LIN {X -0.362,Y -583.040,Z 935.630,A 0.000,B 0.000,C 90.000,E1 149.410} C_DIS
LIN {X -0.117,Y -588.452,Z 935.622,A 0.000,B 0.000,C 90.000,E1 148.043} C_DIS
LIN {X 0.030,Y -592.572,Z 935.617,A 0.000,B 0.000,C 90.000,E1 146.962} C_DIS
LIN {X 0.227,Y -596.675,Z 935.611,A 0.000,B 0.000,C 90.000,E1 145.881} C_DIS
LIN {X 0.218,Y -601.491,Z 935.603,A 0.000,B 0.000,C 90.000,E1 144.562} C_DIS
LIN {X -0.105,Y -605.216,Z 935.597,A 0.000,B 0.000,C 90.000,E1 143.543} C_DIS
LIN {X -0.187,Y -610.766,Z 935.589,A 0.000,B 0.000,C 90.000,E1 141.984} C_DIS
LIN {X -0.091,Y -615.489,Z 935.582,A 0.000,B 0.000,C 90.000,E1 140.678} C_DIS
LIN {X 0.004,Y -620.250,Z 935.574,A 0.000,B 0.000,C 90.000,E1 139.380} C_DIS
LIN {X 0.191,Y -624.987,Z 935.567,A 0.000,B 0.000,C 90.000,E1 138.081} C_DIS
LIN {X 0.103,Y -633.010,Z 935.556,A 0.000,B 0.000,C 90.000,E1 136.053} C_DIS
LIN {X -0.067,Y -638.812,Z 935.548,A 0.000,B 0.000,C 90.000,E1 134.555} C_DIS
LIN {X -0.121,Y -644.569,Z 935.539,A 0.000,B 0.000,C 90.000,E1 133.056} C_DIS
LIN {X -0.071,Y -651.286,Z 935.530,A 0.000,B 0.000,C 90.000,E1 131.310} C_DIS
LIN {X -0.269,Y -656.035,Z 935.523,A 0.000,B 0.000,C 90.000,E1 130.092} C_DIS
LIN {X 0.143,Y -662.595,Z 935.513,A 0.000,B 0.000,C 90.000,E1 128.338} C_DIS
LIN {X -0.301,Y -667.183,Z 935.506,A 0.000,B 0.000,C 90.000,E1 127.156} C_DIS
LIN {X -0.153,Y -671.681,Z 935.500,A 0.000,B 0.000,C 90.000,E1 125.931} C_DIS
LIN {X 0.096,Y -674.267,Z 935.496,A 0.000,B 0.000,C 90.000,E1 125.185} C_DIS
LIN {X -0.032,Y -678.225,Z 935.489,A 0.000,B 0.000,C 90.000,E1 123.992} C_DIS
LIN {X -0.273,Y -680.447,Z 935.485,A 0.000,B 0.000,C 90.000,E1 123.293} C_DIS
LIN {X -0.309,Y -683.103,Z 935.480,A 0.000,B 0.000,C 90.000,E1 122.339} C_DIS
LIN {X 0.065,Y -684.898,Z 935.476,A 0.000,B 0.000,C 90.000,E1 121.592} C_DIS
LIN {X -0.272,Y -687.033,Z 935.470,A 0.000,B 0.000,C 90.000,E1 120.669} C_DIS
LIN {X 0.137,Y -688.460,Z 935.466,A 0.000,B 0.000,C 90.000,E1 119.922} C_DIS
LIN {X -0.157,Y -690.099,Z 935.461,A 0.000,B 0.000,C 90.000,E1 118.999} C_DIS
LIN {X 0.309,Y -690.840,Z 935.458,A 0.000,B 0.000,C 90.000,E1 118.487} C_DIS
LIN {X -0.282,Y -691.955,Z 935.453,A 0.000,B 0.000,C 90.000,E1 117.590} C_DIS
LIN {X 0.076,Y -692.662,Z 935.448,A 0.000,B 0.000,C 90.000,E1 116.616} C_DIS
LIN {X 0.133,Y -692.971,Z 935.443,A 0.000,B 0.000,C 90.000,E1 115.668} C_DIS
LIN {X 0.198,Y -693.012,Z 935.437,A 0.000,B 0.000,C 90.000,E1 114.719} C_DIS
LIN {X 0.017,Y -692.878,Z 935.434,A 0.000,B 0.000,C 90.000,E1 114.027} C_DIS
LIN {X 0.261,Y -692.673,Z 935.432,A 0.000,B 0.000,C 90.000,E1 113.770} C_DIS
LIN {X -0.167,Y -691.954,Z 935.430,A 0.000,B 0.000,C 90.000,E1 113.334} C_DIS
LIN {X 0.072,Y -691.188,Z 935.428,A 0.000,B 0.000,C 90.000,E1 113.078} C_DIS
LIN {X 0.307,Y -690.243,Z 935.427,A 0.000,B 0.000,C 90.000,E1 112.823} C_DIS
LIN {X 0.273,Y -689.103,Z 935.426,A 0.000,B 0.000,C 90.000,E1 112.589} C_DIS
LIN {X -0.135,Y -686.943,Z 935.424,A 0.000,B 0.000,C 90.000,E1 112.386} C_DIS
LIN {X -0.277,Y -685.755,Z 935.424,A 0.000,B 0.000,C 90.000,E1 112.280} C_DIS
LIN {X 0.059,Y -682.964,Z 935.422,A 0.000,B 0.000,C 90.000,E1 112.025} C_DIS
LIN {X 0.274,Y -681.246,Z 935.422,A 0.000,B 0.000,C 90.000,E1 111.897} C_DIS
LIN {X -0.208,Y -678.934,Z 935.421,A 0.000,B 0.000,C 90.000,E1 111.844} C_DIS
LIN {X 0.195,Y -676.175,Z 935.421,A 0.000,B 0.000,C 90.000,E1 111.716} C_DIS
LIN {X 0.326,Y -671.403,Z 935.420,A 0.000,B 0.000,C 90.000,E1 111.589} C_DIS
LIN {X 0.190,Y -668.015,Z 935.420,A 0.000,B 0.000,C 90.000,E1 111.535} C_DIS
LIN {X -0.330,Y -660.119,Z 935.420,A 0.000,B 0.000,C 90.000,E1 111.535} C_DIS
LIN {X -0.363,Y -639.191,Z 935.419,A 0.000,B 0.000,C 90.000,E1 111.535} C_DIS
LIN {X 0.038,Y -634.303,Z 935.419,A 0.000,B 0.000,C 90.000,E1 111.461} C_DIS
LIN {X -0.248,Y -628.865,Z 935.419,A 0.000,B 0.000,C 90.000,E1 111.408} C_DIS
LIN {X 0.128,Y -621.355,Z 935.418,A 0.000,B 0.000,C 90.000,E1 111.227} C_DIS
LIN {X 0.020,Y -614.885,Z 935.417,A 0.000,B 0.000,C 90.000,E1 111.046} C_DIS
LIN {X -0.101,Y -607.904,Z 935.416,A 0.000,B 0.000,C 90.000,E1 110.791} C_DIS
LIN {X -0.152,Y -602.249,Z 935.414,A 0.000,B 0.000,C 90.000,E1 110.536} C_DIS
LIN {X 0.285,Y -595.632,Z 935.412,A 0.000,B 0.000,C 90.000,E1 110.120} C_DIS
LIN {X -0.258,Y -586.968,Z 935.409,A 0.000,B 0.000,C 90.000,E1 109.577} C_DIS
LIN {X 0.123,Y -577.996,Z 935.405,A 0.000,B 0.000,C 90.000,E1 108.906} C_DIS
LIN {X -0.168,Y -569.590,Z 935.403,A 0.000,B 0.000,C 90.000,E1 108.471} C_DIS
LIN {X 0.206,Y -564.053,Z 935.401,A 0.000,B 0.000,C 90.000,E1 108.181} C_DIS
LIN {X -0.172,Y -558.813,Z 935.400,A 0.000,B 0.000,C 90.000,E1 108.000} C_DIS
LIN {X 0.052,Y -554.272,Z 935.399,A 0.000,B 0.000,C 90.000,E1 107.764} C_DIS
LIN {X 0.127,Y -552.298,Z 935.398,A 0.000,B 0.000,C 90.000,E1 107.583} C_DIS
LIN {X 0.089,Y -552.284,Z 935.398,A 0.000,B 0.000,C 90.000,E1 107.583} C_DIS
LIN {X -0.183,Y -551.902,Z 935.397,A 0.000,B 0.000,C 90.000,E1 107.402} C_DIS
LIN {X 0.198,Y -552.578,Z 935.387,A 0.000,B 0.000,C 90.000,E1 105.552} C_DIS
LIN {X 0.228,Y -553.493,Z 935.376,A 0.000,B 0.000,C 90.000,E1 103.592} C_DIS
LIN {X 0.150,Y -554.878,Z 935.363,A 0.000,B 0.000,C 90.000,E1 101.366} C_DIS
LIN {X -0.122,Y -556.475,Z 935.352,A 0.000,B 0.000,C 90.000,E1 99.443} C_DIS
LIN {X 0.047,Y -557.835,Z 935.343,A 0.000,B 0.000,C 90.000,E1 97.757} C_DIS
LIN {X 0.020,Y -558.827,Z 935.335,A 0.000,B 0.000,C 90.000,E1 96.372} C_DIS
LIN {X -0.047,Y -559.704,Z 935.328,A 0.000,B 0.000,C 90.000,E1 94.992} C_DIS
LIN {X -0.006,Y -560.667,Z 935.319,A 0.000,B 0.000,C 90.000,E1 93.326} C_DIS
LIN {X -0.166,Y -561.192,Z 935.312,A 0.000,B 0.000,C 90.000,E1 92.236} C_DIS
LIN {X -0.226,Y -561.817,Z 935.305,A 0.000,B 0.000,C 90.000,E1 90.859} C_DIS
LIN {X 0.174,Y -562.176,Z 935.299,A 0.000,B 0.000,C 90.000,E1 89.714} C_DIS
LIN {X 0.114,Y -562.543,Z 935.291,A 0.000,B 0.000,C 90.000,E1 88.339} C_DIS
LIN {X 0.072,Y -562.878,Z 935.283,A 0.000,B 0.000,C 90.000,E1 86.963} C_DIS
LIN {X -0.254,Y -563.186,Z 935.272,A 0.000,B 0.000,C 90.000,E1 85.065} C_DIS
LIN {X -0.244,Y -563.359,Z 935.265,A 0.000,B 0.000,C 90.000,E1 83.685} C_DIS
LIN {X -0.175,Y -563.591,Z 935.257,A 0.000,B 0.000,C 90.000,E1 82.299} C_DIS
LIN {X 0.054,Y -564.071,Z 935.248,A 0.000,B 0.000,C 90.000,E1 80.622} C_DIS
LIN {X 0.152,Y -564.952,Z 935.236,A 0.000,B 0.000,C 90.000,E1 78.409} C_DIS
LIN {X -0.203,Y -566.027,Z 935.225,A 0.000,B 0.000,C 90.000,E1 76.520} C_DIS
LIN {X -0.077,Y -566.750,Z 935.219,A 0.000,B 0.000,C 90.000,E1 75.408} C_DIS
LIN {X 0.137,Y -567.695,Z 935.210,A 0.000,B 0.000,C 90.000,E1 73.740} C_DIS
LIN {X -0.175,Y -568.620,Z 935.201,A 0.000,B 0.000,C 90.000,E1 72.127} C_DIS
LIN {X 0.043,Y -569.522,Z 935.190,A 0.000,B 0.000,C 90.000,E1 70.188} C_DIS
LIN {X 0.125,Y -570.063,Z 935.181,A 0.000,B 0.000,C 90.000,E1 68.539} C_DIS
LIN {X 0.249,Y -570.504,Z 935.170,A 0.000,B 0.000,C 90.000,E1 66.613} C_DIS
LIN {X 0.085,Y -570.711,Z 935.164,A 0.000,B 0.000,C 90.000,E1 65.537} C_DIS
LIN {X -0.070,Y -570.859,Z 935.158,A 0.000,B 0.000,C 90.000,E1 64.460} C_DIS
LIN {X -0.227,Y -571.063,Z 935.152,A 0.000,B 0.000,C 90.000,E1 63.384} C_DIS
LIN {X 0.211,Y -571.167,Z 935.144,A 0.000,B 0.000,C 90.000,E1 61.975} C_DIS
LIN {X 0.247,Y -571.113,Z 935.135,A 0.000,B 0.000,C 90.000,E1 60.333} C_DIS
LIN {X -0.038,Y -571.169,Z 935.128,A 0.000,B 0.000,C 90.000,E1 58.997} C_DIS
LIN {X -0.267,Y -571.086,Z 935.123,A 0.000,B 0.000,C 90.000,E1 58.201} C_DIS
LIN {X -0.310,Y -570.565,Z 935.113,A 0.000,B 0.000,C 90.000,E1 56.294} C_DIS
LIN {X 0.015,Y -569.854,Z 935.105,A 0.000,B 0.000,C 90.000,E1 54.895} C_DIS
LIN {X -0.133,Y -569.057,Z 935.097,A 0.000,B 0.000,C 90.000,E1 53.543} C_DIS
LIN {X -0.094,Y -568.344,Z 935.093,A 0.000,B 0.000,C 90.000,E1 52.718} C_DIS
LIN {X -0.174,Y -567.529,Z 935.088,A 0.000,B 0.000,C 90.000,E1 51.904} C_DIS
LIN {X -0.139,Y -566.224,Z 935.082,A 0.000,B 0.000,C 90.000,E1 50.803} C_DIS
LIN {X -0.237,Y -565.126,Z 935.078,A 0.000,B 0.000,C 90.000,E1 49.989} C_DIS
LIN {X 0.344,Y -564.350,Z 935.075,A 0.000,B 0.000,C 90.000,E1 49.380} C_DIS
LIN {X -0.201,Y -562.938,Z 935.070,A 0.000,B 0.000,C 90.000,E1 48.609} C_DIS
LIN {X 0.125,Y -560.668,Z 935.064,A 0.000,B 0.000,C 90.000,E1 47.472} C_DIS
LIN {X -0.124,Y -559.464,Z 935.061,A 0.000,B 0.000,C 90.000,E1 46.944} C_DIS
LIN {X 0.117,Y -556.574,Z 935.055,A 0.000,B 0.000,C 90.000,E1 45.810} C_DIS
LIN {X -0.221,Y -555.832,Z 935.053,A 0.000,B 0.000,C 90.000,E1 45.567} C_DIS
LIN {X -0.027,Y -552.309,Z 935.047,A 0.000,B 0.000,C 90.000,E1 44.433} C_DIS
LIN {X 0.007,Y -551.392,Z 935.045,A 0.000,B 0.000,C 90.000,E1 44.150} C_DIS
LIN {X 0.109,Y -548.247,Z 935.041,A 0.000,B 0.000,C 90.000,E1 43.299} C_DIS
LIN {X -0.220,Y -546.013,Z 935.038,A 0.000,B 0.000,C 90.000,E1 42.771} C_DIS
LIN {X 0.002,Y -542.942,Z 935.034,A 0.000,B 0.000,C 90.000,E1 42.043} C_DIS
LIN {X 0.230,Y -539.518,Z 935.030,A 0.000,B 0.000,C 90.000,E1 41.310} C_DIS
LIN {X -0.153,Y -536.559,Z 935.027,A 0.000,B 0.000,C 90.000,E1 40.782} C_DIS
LIN {X 0.198,Y -533.440,Z 935.023,A 0.000,B 0.000,C 90.000,E1 40.172} C_DIS
LIN {X -0.225,Y -530.096,Z 935.020,A 0.000,B 0.000,C 90.000,E1 39.644} C_DIS
LIN {X 0.010,Y -523.010,Z 935.014,A 0.000,B 0.000,C 90.000,E1 38.463} C_DIS
LIN {X 0.059,Y -518.243,Z 935.010,A 0.000,B 0.000,C 90.000,E1 37.729} C_DIS
LIN {X -0.127,Y -512.183,Z 935.005,A 0.000,B 0.000,C 90.000,E1 36.870} C_DIS
LIN {X 0.229,Y -506.756,Z 935.001,A 0.000,B 0.000,C 90.000,E1 36.091} C_DIS
LIN {X -0.065,Y -503.303,Z 934.998,A 0.000,B 0.000,C 90.000,E1 35.678} C_DIS
LIN {X 0.155,Y -500.020,Z 934.996,A 0.000,B 0.000,C 90.000,E1 35.231} C_DIS
LIN {X 0.123,Y -493.520,Z 934.992,A 0.000,B 0.000,C 90.000,E1 34.485} C_DIS
LIN {X 0.010,Y -490.928,Z 934.990,A 0.000,B 0.000,C 90.000,E1 34.199} C_DIS
LIN {X -0.230,Y -483.914,Z 934.986,A 0.000,B 0.000,C 90.000,E1 33.499} C_DIS
LIN {X 0.225,Y -478.200,Z 934.983,A 0.000,B 0.000,C 90.000,E1 32.880} C_DIS
LIN {X 0.050,Y -470.972,Z 934.979,A 0.000,B 0.000,C 90.000,E1 32.212} C_DIS
LIN {X 0.072,Y -460.714,Z 934.974,A 0.000,B 0.000,C 90.000,E1 31.288} C_DIS
LIN {X -0.009,Y -450.031,Z 934.969,A 0.000,B 0.000,C 90.000,E1 30.384} C_DIS
LIN {X 0.134,Y -437.697,Z 934.963,A 0.000,B 0.000,C 90.000,E1 29.333} C_DIS
LIN {X 0.113,Y -416.401,Z 934.953,A 0.000,B 0.000,C 90.000,E1 27.462} C_DIS
LIN {X -0.085,Y -400.384,Z 934.944,A 0.000,B 0.000,C 90.000,E1 25.924} C_DIS
LIN {X 0.089,Y -397.514,Z 934.942,A 0.000,B 0.000,C 90.000,E1 25.591} C_DIS
LIN {X -0.048,Y -393.296,Z 934.939,A 0.000,B 0.000,C 90.000,E1 25.027} C_DIS
LIN {X -0.019,Y -390.739,Z 934.936,A 0.000,B 0.000,C 90.000,E1 24.515} C_DIS
LIN {X -0.019,Y -389.495,Z 934.934,A 0.000,B 0.000,C 90.000,E1 24.027} C_DIS
LIN {X 0.106,Y -388.958,Z 934.929,A 0.000,B 0.000,C 90.000,E1 23.206} C_DIS
LIN {X -0.027,Y -389.146,Z 934.924,A 0.000,B 0.000,C 90.000,E1 22.333} C_DIS
LIN {X -0.081,Y -392.397,Z 934.904,A 0.000,B 0.000,C 90.000,E1 18.779} C_DIS
LIN {X 0.180,Y -395.235,Z 934.891,A 0.000,B 0.000,C 90.000,E1 16.260} C_DIS
LIN {X -0.033,Y -399.362,Z 934.873,A 0.000,B 0.000,C 90.000,E1 13.119} C_DIS
LIN {X 0.028,Y -403.553,Z 934.857,A 0.000,B 0.000,C 90.000,E1 10.310} C_DIS
LIN {X 0.037,Y -405.864,Z 934.850,A 0.000,B 0.000,C 90.000,E1 8.916} C_DIS
LIN {X 0.060,Y -409.516,Z 934.838,A 0.000,B 0.000,C 90.000,E1 6.834} C_DIS
LIN {X 0.117,Y -414.812,Z 934.823,A 0.000,B 0.000,C 90.000,E1 4.073} C_DIS
LIN {X -0.069,Y -421.450,Z 934.806,A 0.000,B 0.000,C 90.000,E1 1.031} C_DIS
LIN {X -0.163,Y -426.045,Z 934.795,A 0.000,B 0.000,C 90.000,E1 359.141} C_DIS
LIN {X -0.053,Y -427.988,Z 934.791,A 0.000,B 0.000,C 90.000,E1 358.453} C_DIS
LIN {X 0.173,Y -430.450,Z 934.788,A 0.000,B 0.000,C 90.000,E1 357.764} C_DIS
LIN {X 0.208,Y -431.327,Z 934.787,A 0.000,B 0.000,C 90.000,E1 357.593} C_DIS
LIN {X -0.150,Y -433.776,Z 934.785,A 0.000,B 0.000,C 90.000,E1 357.306} C_DIS
LIN {X 0.127,Y -435.457,Z 934.784,A 0.000,B 0.000,C 90.000,E1 357.020} C_DIS
LIN {X -0.069,Y -436.183,Z 934.783,A 0.000,B 0.000,C 90.000,E1 356.963} C_DIS
LIN {X -0.052,Y -441.451,Z 934.781,A 0.000,B 0.000,C 90.000,E1 356.560} C_DIS
LIN {X 0.217,Y -447.579,Z 934.779,A 0.000,B 0.000,C 90.000,E1 356.216} C_DIS
LIN {X 0.059,Y -454.281,Z 934.777,A 0.000,B 0.000,C 90.000,E1 355.927} C_DIS
LIN {X 0.204,Y -467.603,Z 934.774,A 0.000,B 0.000,C 90.000,E1 355.241} C_DIS
LIN {X 0.040,Y -482.471,Z 934.769,A 0.000,B 0.000,C 90.000,E1 354.489} C_DIS
LIN {X -0.188,Y -490.646,Z 934.767,A 0.000,B 0.000,C 90.000,E1 354.090} C_DIS
LIN {X 0.143,Y -503.360,Z 934.763,A 0.000,B 0.000,C 90.000,E1 353.337} C_DIS
LIN {X 0.162,Y -512.995,Z 934.760,A 0.000,B 0.000,C 90.000,E1 352.761} C_DIS
LIN {X -0.105,Y -522.411,Z 934.757,A 0.000,B 0.000,C 90.000,E1 352.186} C_DIS
LIN {X 0.229,Y -528.534,Z 934.754,A 0.000,B 0.000,C 90.000,E1 351.724} C_DIS
LIN {X -0.112,Y -535.939,Z 934.751,A 0.000,B 0.000,C 90.000,E1 351.197} C_DIS
LIN {X -0.284,Y -543.099,Z 934.748,A 0.000,B 0.000,C 90.000,E1 350.622} C_DIS
LIN {X -0.120,Y -549.902,Z 934.744,A 0.000,B 0.000,C 90.000,E1 349.982} C_DIS
LIN {X -0.031,Y -555.068,Z 934.741,A 0.000,B 0.000,C 90.000,E1 349.454} C_DIS
LIN {X 0.254,Y -561.010,Z 934.738,A 0.000,B 0.000,C 90.000,E1 348.757} C_DIS
LIN {X 0.045,Y -568.927,Z 934.732,A 0.000,B 0.000,C 90.000,E1 347.813} C_DIS
LIN {X 0.167,Y -573.969,Z 934.729,A 0.000,B 0.000,C 90.000,E1 347.117} C_DIS
LIN {X 0.219,Y -579.696,Z 934.724,A 0.000,B 0.000,C 90.000,E1 346.297} C_DIS
LIN {X -0.001,Y -583.991,Z 934.720,A 0.000,B 0.000,C 90.000,E1 345.644} C_DIS
LIN {X 0.301,Y -588.909,Z 934.716,A 0.000,B 0.000,C 90.000,E1 344.810} C_DIS
LIN {X -0.146,Y -594.211,Z 934.711,A 0.000,B 0.000,C 90.000,E1 343.921} C_DIS
LIN {X -0.028,Y -599.726,Z 934.705,A 0.000,B 0.000,C 90.000,E1 342.851} C_DIS
LIN {X -0.052,Y -608.018,Z 934.695,A 0.000,B 0.000,C 90.000,E1 341.148} C_DIS
LIN {X -0.108,Y -612.243,Z 934.690,A 0.000,B 0.000,C 90.000,E1 340.242} C_DIS
LIN {X -0.176,Y -617.810,Z 934.683,A 0.000,B 0.000,C 90.000,E1 338.954} C_DIS
LIN {X -0.155,Y -622.956,Z 934.676,A 0.000,B 0.000,C 90.000,E1 337.667} C_DIS
LIN {X 0.171,Y -625.871,Z 934.672,A 0.000,B 0.000,C 90.000,E1 336.869} C_DIS
LIN {X -0.037,Y -629.434,Z 934.666,A 0.000,B 0.000,C 90.000,E1 335.869} C_DIS
LIN {X 0.034,Y -632.073,Z 934.662,A 0.000,B 0.000,C 90.000,E1 335.101} C_DIS
LIN {X 0.181,Y -635.351,Z 934.656,A 0.000,B 0.000,C 90.000,E1 334.076} C_DIS
LIN {X 0.141,Y -639.086,Z 934.649,A 0.000,B 0.000,C 90.000,E1 332.820} C_DIS
LIN {X -0.192,Y -641.900,Z 934.644,A 0.000,B 0.000,C 90.000,E1 331.847} C_DIS
LIN {X -0.177,Y -644.440,Z 934.638,A 0.000,B 0.000,C 90.000,E1 330.845} C_DIS
LIN {X 0.042,Y -647.954,Z 934.630,A 0.000,B 0.000,C 90.000,E1 329.331} C_DIS
LIN {X 0.148,Y -650.027,Z 934.624,A 0.000,B 0.000,C 90.000,E1 328.329} C_DIS
LIN {X -0.271,Y -651.825,Z 934.619,A 0.000,B 0.000,C 90.000,E1 327.375} C_DIS
LIN {X -0.209,Y -653.092,Z 934.615,A 0.000,B 0.000,C 90.000,E1 326.628} C_DIS
LIN {X 0.314,Y -654.556,Z 934.609,A 0.000,B 0.000,C 90.000,E1 325.595} C_DIS
LIN {X 0.327,Y -656.333,Z 934.601,A 0.000,B 0.000,C 90.000,E1 324.116} C_DIS
LIN {X 0.354,Y -657.418,Z 934.595,A 0.000,B 0.000,C 90.000,E1 323.130} C_DIS
LIN {X -0.117,Y -658.660,Z 934.587,A 0.000,B 0.000,C 90.000,E1 321.698} C_DIS
LIN {X -0.230,Y -660.230,Z 934.576,A 0.000,B 0.000,C 90.000,E1 319.747} C_DIS
LIN {X 0.161,Y -661.603,Z 934.567,A 0.000,B 0.000,C 90.000,E1 318.000} C_DIS
LIN {X 0.130,Y -662.427,Z 934.561,A 0.000,B 0.000,C 90.000,E1 317.025} C_DIS
LIN {X 0.063,Y -663.474,Z 934.555,A 0.000,B 0.000,C 90.000,E1 315.810} C_DIS
LIN {X -0.018,Y -665.725,Z 934.540,A 0.000,B 0.000,C 90.000,E1 313.137} C_DIS
LIN {X -0.002,Y -667.109,Z 934.532,A 0.000,B 0.000,C 90.000,E1 311.676} C_DIS
LIN {X 0.115,Y -668.674,Z 934.522,A 0.000,B 0.000,C 90.000,E1 309.967} C_DIS
LIN {X 0.185,Y -669.760,Z 934.515,A 0.000,B 0.000,C 90.000,E1 308.749} C_DIS
LIN {X -0.163,Y -670.700,Z 934.509,A 0.000,B 0.000,C 90.000,E1 307.569} C_DIS
LIN {X 0.044,Y -671.266,Z 934.503,A 0.000,B 0.000,C 90.000,E1 306.583} C_DIS
LIN {X -0.258,Y -671.525,Z 934.499,A 0.000,B 0.000,C 90.000,E1 305.884} C_DIS
LIN {X -0.326,Y -672.092,Z 934.490,A 0.000,B 0.000,C 90.000,E1 304.199} C_DIS
LIN {X -0.084,Y -673.147,Z 934.478,A 0.000,B 0.000,C 90.000,E1 302.005} C_DIS
LIN {X -0.300,Y -678.749,Z 934.447,A 0.000,B 0.000,C 90.000,E1 296.488} C_DIS
LIN {X -0.219,Y -680.724,Z 934.440,A 0.000,B 0.000,C 90.000,E1 295.283} C_DIS
LIN {X -0.106,Y -682.529,Z 934.434,A 0.000,B 0.000,C 90.000,E1 294.079} C_DIS
LIN {X 0.238,Y -683.405,Z 934.430,A 0.000,B 0.000,C 90.000,E1 293.334} C_DIS
LIN {X -0.184,Y -683.659,Z 934.428,A 0.000,B 0.000,C 90.000,E1 293.131} C_DIS
LIN {X -0.037,Y -683.885,Z 934.426,A 0.000,B 0.000,C 90.000,E1 292.642} C_DIS
LIN {X 0.168,Y -683.807,Z 934.424,A 0.000,B 0.000,C 90.000,E1 292.386} C_DIS
LIN {X 0.318,Y -683.227,Z 934.422,A 0.000,B 0.000,C 90.000,E1 291.897} C_DIS
LIN {X -0.367,Y -682.487,Z 934.421,A 0.000,B 0.000,C 90.000,E1 291.716} C_DIS
LIN {X -0.266,Y -681.729,Z 934.420,A 0.000,B 0.000,C 90.000,E1 291.589} C_DIS
LIN {X -0.127,Y -677.804,Z 934.417,A 0.000,B 0.000,C 90.000,E1 291.099} C_DIS
LIN {X -0.035,Y -676.505,Z 934.417,A 0.000,B 0.000,C 90.000,E1 290.972} C_DIS
LIN {X 0.005,Y -669.890,Z 934.414,A 0.000,B 0.000,C 90.000,E1 290.556} C_DIS
LIN {X 0.263,Y -663.844,Z 934.412,A 0.000,B 0.000,C 90.000,E1 290.174} C_DIS
LIN {X -0.173,Y -662.168,Z 934.411,A 0.000,B 0.000,C 90.000,E1 290.066} C_DIS
LIN {X -0.213,Y -662.151,Z 934.411,A 0.000,B 0.000,C 90.000,E1 290.066} C_DIS
LIN {X -0.036,Y -661.882,Z 934.411,A 0.000,B 0.000,C 90.000,E1 289.939} C_DIS
LIN {X 0.111,Y -661.958,Z 934.410,A 0.000,B 0.000,C 90.000,E1 289.812} C_DIS
LIN {X 0.003,Y -662.374,Z 934.409,A 0.000,B 0.000,C 90.000,E1 289.577} C_DIS
LIN {X 0.118,Y -663.165,Z 934.407,A 0.000,B 0.000,C 90.000,E1 289.322} C_DIS
LIN {X 0.016,Y -664.110,Z 934.406,A 0.000,B 0.000,C 90.000,E1 289.087} C_DIS
LIN {X 0.010,Y -667.041,Z 934.403,A 0.000,B 0.000,C 90.000,E1 288.489} C_DIS
LIN {X 0.037,Y -671.497,Z 934.398,A 0.000,B 0.000,C 90.000,E1 287.638} C_DIS
LIN {X -0.101,Y -673.850,Z 934.395,A 0.000,B 0.000,C 90.000,E1 287.166} C_DIS
LIN {X -0.081,Y -676.901,Z 934.391,A 0.000,B 0.000,C 90.000,E1 286.441} C_DIS
LIN {X -0.041,Y -679.329,Z 934.387,A 0.000,B 0.000,C 90.000,E1 285.717} C_DIS
LIN {X -0.125,Y -680.682,Z 934.385,A 0.000,B 0.000,C 90.000,E1 285.245} C_DIS
LIN {X -0.262,Y -682.869,Z 934.379,A 0.000,B 0.000,C 90.000,E1 284.300} C_DIS
LIN {X -0.320,Y -683.809,Z 934.377,A 0.000,B 0.000,C 90.000,E1 283.828} C_DIS
LIN {X 0.250,Y -685.364,Z 934.371,A 0.000,B 0.000,C 90.000,E1 282.827} C_DIS
LIN {X 0.187,Y -686.270,Z 934.367,A 0.000,B 0.000,C 90.000,E1 282.119} C_DIS
LIN {X 0.008,Y -686.722,Z 934.365,A 0.000,B 0.000,C 90.000,E1 281.658} C_DIS
LIN {X -0.029,Y -686.947,Z 934.362,A 0.000,B 0.000,C 90.000,E1 281.186} C_DIS
LIN {X -0.067,Y -686.915,Z 934.360,A 0.000,B 0.000,C 90.000,E1 280.715} C_DIS
LIN {X -0.233,Y -686.522,Z 934.357,A 0.000,B 0.000,C 90.000,E1 280.254} C_DIS
LIN {X -0.255,Y -686.208,Z 934.356,A 0.000,B 0.000,C 90.000,E1 280.018} C_DIS
LIN {X 0.256,Y -685.292,Z 934.353,A 0.000,B 0.000,C 90.000,E1 279.500} C_DIS
LIN {X 0.197,Y -683.887,Z 934.350,A 0.000,B 0.000,C 90.000,E1 279.029} C_DIS
LIN {X 0.020,Y -682.123,Z 934.348,A 0.000,B 0.000,C 90.000,E1 278.568} C_DIS
LIN {X -0.163,Y -679.996,Z 934.345,A 0.000,B 0.000,C 90.000,E1 278.106} C_DIS
LIN {X 0.181,Y -675.839,Z 934.340,A 0.000,B 0.000,C 90.000,E1 277.239} C_DIS
LIN {X -0.280,Y -670.704,Z 934.335,A 0.000,B 0.000,C 90.000,E1 276.315} C_DIS
LIN {X 0.129,Y -667.800,Z 934.332,A 0.000,B 0.000,C 90.000,E1 275.796} C_DIS
LIN {X -0.146,Y -664.503,Z 934.330,A 0.000,B 0.000,C 90.000,E1 275.334} C_DIS
LIN {X 0.123,Y -659.733,Z 934.326,A 0.000,B 0.000,C 90.000,E1 274.702} C_DIS
LIN {X -0.254,Y -655.607,Z 934.323,A 0.000,B 0.000,C 90.000,E1 274.245} C_DIS
LIN {X -0.060,Y -649.876,Z 934.320,A 0.000,B 0.000,C 90.000,E1 273.612} C_DIS
LIN {X 0.281,Y -645.013,Z 934.317,A 0.000,B 0.000,C 90.000,E1 273.094} C_DIS
LIN {X 0.109,Y -638.445,Z 934.314,A 0.000,B 0.000,C 90.000,E1 272.522} C_DIS
LIN {X 0.273,Y -631.457,Z 934.311,A 0.000,B 0.000,C 90.000,E1 271.949} C_DIS
LIN {X 0.211,Y -624.054,Z 934.308,A 0.000,B 0.000,C 90.000,E1 271.432} C_DIS
LIN {X 0.212,Y -617.936,Z 934.306,A 0.000,B 0.000,C 90.000,E1 271.031} C_DIS
LIN {X -0.205,Y -611.553,Z 934.304,A 0.000,B 0.000,C 90.000,E1 270.688} C_DIS
LIN {X 0.261,Y -604.962,Z 934.302,A 0.000,B 0.000,C 90.000,E1 270.286} C_DIS
LIN {X -0.198,Y -598.161,Z 934.300,A 0.000,B 0.000,C 90.000,E1 270.000} C_DIS
LIN {X 0.219,Y -591.125,Z 934.298,A 0.000,B 0.000,C 90.000,E1 269.656} C_DIS
LIN {X -0.142,Y -585.444,Z 934.297,A 0.000,B 0.000,C 90.000,E1 269.484} C_DIS
LIN {X -0.137,Y -577.860,Z 934.296,A 0.000,B 0.000,C 90.000,E1 269.255} C_DIS
LIN {X -0.221,Y -570.064,Z 934.295,A 0.000,B 0.000,C 90.000,E1 269.083} C_DIS
LIN {X -0.193,Y -563.989,Z 934.294,A 0.000,B 0.000,C 90.000,E1 268.969} C_DIS
LIN {X -0.243,Y -557.682,Z 934.294,A 0.000,B 0.000,C 90.000,E1 268.912} C_DIS
LIN {X -0.093,Y -552.004,Z 934.294,A 0.000,B 0.000,C 90.000,E1 268.854} C_DIS
LIN {X 0.239,Y -550.919,Z 934.294,A 0.000,B 0.000,C 90.000,E1 268.797} C_DIS
LIN {X 0.193,Y -550.707,Z 934.293,A 0.000,B 0.000,C 90.000,E1 268.797} C_DIS
LIN {X -0.185,Y -549.196,Z 934.292,A 0.000,B 0.000,C 90.000,E1 268.625} C_DIS
LIN {X 0.184,Y -545.518,Z 934.290,A 0.000,B 0.000,C 90.000,E1 268.165} C_DIS
LIN {X 0.060,Y -544.029,Z 934.289,A 0.000,B 0.000,C 90.000,E1 268.051} C_DIS
LIN {X 0.017,Y -543.977,Z 934.289,A 0.000,B 0.000,C 90.000,E1 268.051} C_DIS
LIN {X 0.228,Y -543.627,Z 934.288,A 0.000,B 0.000,C 90.000,E1 267.879} C_DIS
LIN {X -0.146,Y -542.881,Z 934.285,A 0.000,B 0.000,C 90.000,E1 267.364} C_DIS
LIN {X 0.213,Y -540.432,Z 934.270,A 0.000,B 0.000,C 90.000,E1 264.489} C_DIS
LIN {X -0.119,Y -539.299,Z 934.260,A 0.000,B 0.000,C 90.000,E1 262.818} C_DIS
LIN {X 0.055,Y -538.331,Z 934.252,A 0.000,B 0.000,C 90.000,E1 261.376} C_DIS
LIN {X 0.249,Y -537.661,Z 934.247,A 0.000,B 0.000,C 90.000,E1 260.500} C_DIS
LIN {X -0.182,Y -536.656,Z 934.243,A 0.000,B 0.000,C 90.000,E1 259.690} C_DIS
LIN {X 0.056,Y -535.034,Z 934.236,A 0.000,B 0.000,C 90.000,E1 258.522} C_DIS
LIN {X 0.172,Y -530.972,Z 934.219,A 0.000,B 0.000,C 90.000,E1 255.353} C_DIS
LIN {X 0.117,Y -528.945,Z 934.209,A 0.000,B 0.000,C 90.000,E1 253.630} C_DIS
LIN {X 0.166,Y -526.789,Z 934.200,A 0.000,B 0.000,C 90.000,E1 251.891} C_DIS
LIN {X -0.163,Y -524.571,Z 934.190,A 0.000,B 0.000,C 90.000,E1 250.188} C_DIS
LIN {X -0.022,Y -522.711,Z 934.182,A 0.000,B 0.000,C 90.000,E1 248.720} C_DIS
LIN {X 0.277,Y -520.814,Z 934.174,A 0.000,B 0.000,C 90.000,E1 247.230} C_DIS
LIN {X 0.204,Y -518.179,Z 934.164,A 0.000,B 0.000,C 90.000,E1 245.485} C_DIS
LIN {X -0.183,Y -515.465,Z 934.154,A 0.000,B 0.000,C 90.000,E1 243.768} C_DIS
LIN {X -0.049,Y -513.030,Z 934.146,A 0.000,B 0.000,C 90.000,E1 242.281} C_DIS
LIN {X 0.038,Y -510.576,Z 934.138,A 0.000,B 0.000,C 90.000,E1 240.795} C_DIS
LIN {X -0.011,Y -508.509,Z 934.131,A 0.000,B 0.000,C 90.000,E1 239.616} C_DIS
LIN {X 0.164,Y -506.356,Z 934.125,A 0.000,B 0.000,C 90.000,E1 238.408} C_DIS
LIN {X -0.120,Y -503.875,Z 934.118,A 0.000,B 0.000,C 90.000,E1 237.248} C_DIS
LIN {X -0.264,Y -499.775,Z 934.108,A 0.000,B 0.000,C 90.000,E1 235.468} C_DIS
LIN {X -0.204,Y -494.327,Z 934.095,A 0.000,B 0.000,C 90.000,E1 233.050} C_DIS
LIN {X -0.235,Y -491.067,Z 934.086,A 0.000,B 0.000,C 90.000,E1 231.537} C_DIS
LIN {X -0.027,Y -487.673,Z 934.078,A 0.000,B 0.000,C 90.000,E1 229.989} C_DIS
LIN {X -0.123,Y -483.469,Z 934.068,A 0.000,B 0.000,C 90.000,E1 228.162} C_DIS
LIN {X 0.131,Y -478.613,Z 934.056,A 0.000,B 0.000,C 90.000,E1 225.972} C_DIS
LIN {X 0.030,Y -475.242,Z 934.047,A 0.000,B 0.000,C 90.000,E1 224.433} C_DIS
LIN {X 0.297,Y -471.084,Z 934.036,A 0.000,B 0.000,C 90.000,E1 222.528} C_DIS
LIN {X 0.070,Y -467.583,Z 934.028,A 0.000,B 0.000,C 90.000,E1 220.987} C_DIS
LIN {X 0.038,Y -462.161,Z 934.014,A 0.000,B 0.000,C 90.000,E1 218.463} C_DIS
LIN {X -0.046,Y -459.386,Z 934.007,A 0.000,B 0.000,C 90.000,E1 217.202} C_DIS
LIN {X 0.015,Y -455.975,Z 933.998,A 0.000,B 0.000,C 90.000,E1 215.598} C_DIS
LIN {X 0.020,Y -452.484,Z 933.989,A 0.000,B 0.000,C 90.000,E1 213.992} C_DIS
LIN {X -0.061,Y -446.698,Z 933.975,A 0.000,B 0.000,C 90.000,E1 211.416} C_DIS
LIN {X -0.171,Y -443.828,Z 933.967,A 0.000,B 0.000,C 90.000,E1 210.129} C_DIS
LIN {X -0.078,Y -439.583,Z 933.956,A 0.000,B 0.000,C 90.000,E1 208.153} C_DIS
LIN {X 0.044,Y -436.809,Z 933.949,A 0.000,B 0.000,C 90.000,E1 206.821} C_DIS
LIN {X -0.039,Y -432.386,Z 933.938,A 0.000,B 0.000,C 90.000,E1 204.847} C_DIS
LIN {X 0.154,Y -428.022,Z 933.927,A 0.000,B 0.000,C 90.000,E1 202.823} C_DIS
LIN {X -0.103,Y -423.545,Z 933.916,A 0.000,B 0.000,C 90.000,E1 200.844} C_DIS
LIN {X 0.146,Y -417.186,Z 933.899,A 0.000,B 0.000,C 90.000,E1 197.764} C_DIS
LIN {X -0.002,Y -413.844,Z 933.889,A 0.000,B 0.000,C 90.000,E1 196.079} C_DIS
LIN {X -0.067,Y -411.056,Z 933.882,A 0.000,B 0.000,C 90.000,E1 194.717} C_DIS
LIN {X 0.066,Y -404.789,Z 933.865,A 0.000,B 0.000,C 90.000,E1 191.591} C_DIS
LIN {X 0.079,Y -401.420,Z 933.855,A 0.000,B 0.000,C 90.000,E1 189.849} C_DIS
LIN {X 0.009,Y -397.329,Z 933.843,A 0.000,B 0.000,C 90.000,E1 187.757} C_DIS
LIN {X -0.150,Y -394.647,Z 933.835,A 0.000,B 0.000,C 90.000,E1 186.372} C_DIS
LIN {X 0.017,Y -388.684,Z 933.818,A 0.000,B 0.000,C 90.000,E1 183.154} C_DIS
LIN {X -0.067,Y -383.430,Z 933.800,A 0.000,B 0.000,C 90.000,E1 179.943} C_DIS
LIN {X -0.016,Y -382.158,Z 933.794,A 0.000,B 0.000,C 90.000,E1 178.854} C_DIS
LIN {X 0.087,Y -381.481,Z 933.789,A 0.000,B 0.000,C 90.000,E1 177.936} C_DIS
LIN {X 0.132,Y -381.508,Z 933.783,A 0.000,B 0.000,C 90.000,E1 176.963} C_DIS
LIN {X -0.090,Y -382.040,Z 933.779,A 0.000,B 0.000,C 90.000,E1 176.274} C_DIS
LIN {X 0.134,Y -383.143,Z 933.776,A 0.000,B 0.000,C 90.000,E1 175.698} C_DIS
LIN {X -0.148,Y -383.539,Z 933.775,A 0.000,B 0.000,C 90.000,E1 175.469} C_DIS
LIN {X -0.074,Y -385.292,Z 933.772,A 0.000,B 0.000,C 90.000,E1 175.008} C_DIS
LIN {X 0.159,Y -388.872,Z 933.769,A 0.000,B 0.000,C 90.000,E1 174.375} C_DIS
LIN {X 0.105,Y -390.089,Z 933.768,A 0.000,B 0.000,C 90.000,E1 174.204} C_DIS
LIN {X -0.173,Y -394.665,Z 933.765,A 0.000,B 0.000,C 90.000,E1 173.742} C_DIS
LIN {X 0.042,Y -401.204,Z 933.762,A 0.000,B 0.000,C 90.000,E1 173.109} C_DIS
LIN {X -0.112,Y -414.286,Z 933.756,A 0.000,B 0.000,C 90.000,E1 172.129} C_DIS
LIN {X -0.098,Y -429.985,Z 933.749,A 0.000,B 0.000,C 90.000,E1 170.905} C_DIS
LIN {X -0.152,Y -439.190,Z 933.745,A 0.000,B 0.000,C 90.000,E1 170.151} C_DIS
LIN {X -0.068,Y -448.118,Z 933.741,A 0.000,B 0.000,C 90.000,E1 169.342} C_DIS
LIN {X 0.255,Y -458.464,Z 933.735,A 0.000,B 0.000,C 90.000,E1 168.342} C_DIS
LIN {X 0.022,Y -466.782,Z 933.731,A 0.000,B 0.000,C 90.000,E1 167.521} C_DIS
LIN {X -0.139,Y -477.531,Z 933.724,A 0.000,B 0.000,C 90.000,E1 166.353} C_DIS
LIN {X 0.080,Y -485.098,Z 933.719,A 0.000,B 0.000,C 90.000,E1 165.408} C_DIS
LIN {X -0.174,Y -492.693,Z 933.714,A 0.000,B 0.000,C 90.000,E1 164.519} C_DIS
LIN {X 0.004,Y -498.226,Z 933.710,A 0.000,B 0.000,C 90.000,E1 163.740} C_DIS
LIN {X 0.031,Y -504.749,Z 933.705,A 0.000,B 0.000,C 90.000,E1 162.834} C_DIS
LIN {X 0.149,Y -516.914,Z 933.695,A 0.000,B 0.000,C 90.000,E1 161.040} C_DIS
LIN {X 0.069,Y -521.689,Z 933.691,A 0.000,B 0.000,C 90.000,E1 160.315} C_DIS
LIN {X 0.059,Y -531.922,Z 933.682,A 0.000,B 0.000,C 90.000,E1 158.720} C_DIS
LIN {X 0.161,Y -537.223,Z 933.677,A 0.000,B 0.000,C 90.000,E1 157.847} C_DIS
LIN {X 0.084,Y -549.262,Z 933.666,A 0.000,B 0.000,C 90.000,E1 155.869} C_DIS
LIN {X 0.106,Y -552.497,Z 933.663,A 0.000,B 0.000,C 90.000,E1 155.305} C_DIS
LIN {X -0.149,Y -559.468,Z 933.656,A 0.000,B 0.000,C 90.000,E1 154.076} C_DIS
LIN {X 0.152,Y -564.538,Z 933.651,A 0.000,B 0.000,C 90.000,E1 153.076} C_DIS
LIN {X 0.176,Y -569.929,Z 933.644,A 0.000,B 0.000,C 90.000,E1 151.975} C_DIS
LIN {X -0.225,Y -575.091,Z 933.638,A 0.000,B 0.000,C 90.000,E1 150.923} C_DIS
LIN {X 0.245,Y -577.525,Z 933.635,A 0.000,B 0.000,C 90.000,E1 150.333} C_DIS
LIN {X -0.063,Y -582.178,Z 933.629,A 0.000,B 0.000,C 90.000,E1 149.282} C_DIS
LIN {X 0.167,Y -587.646,Z 933.622,A 0.000,B 0.000,C 90.000,E1 147.916} C_DIS
LIN {X 0.300,Y -591.804,Z 933.616,A 0.000,B 0.000,C 90.000,E1 146.834} C_DIS
LIN {X -0.008,Y -595.935,Z 933.610,A 0.000,B 0.000,C 90.000,E1 145.801} C_DIS
LIN {X -0.265,Y -599.898,Z 933.604,A 0.000,B 0.000,C 90.000,E1 144.769} C_DIS
LIN {X -0.126,Y -603.663,Z 933.598,A 0.000,B 0.000,C 90.000,E1 143.703} C_DIS
LIN {X -0.145,Y -608.333,Z 933.591,A 0.000,B 0.000,C 90.000,E1 142.396} C_DIS
LIN {X 0.025,Y -614.999,Z 933.581,A 0.000,B 0.000,C 90.000,E1 140.561} C_DIS
LIN {X -0.278,Y -619.806,Z 933.574,A 0.000,B 0.000,C 90.000,E1 139.299} C_DIS
LIN {X 0.045,Y -623.639,Z 933.568,A 0.000,B 0.000,C 90.000,E1 138.243} C_DIS
LIN {X 0.036,Y -630.642,Z 933.558,A 0.000,B 0.000,C 90.000,E1 136.458} C_DIS
LIN {X 0.032,Y -634.670,Z 933.553,A 0.000,B 0.000,C 90.000,E1 135.445} C_DIS
LIN {X -0.104,Y -640.465,Z 933.544,A 0.000,B 0.000,C 90.000,E1 133.947} C_DIS
LIN {X -0.045,Y -645.294,Z 933.537,A 0.000,B 0.000,C 90.000,E1 132.690} C_DIS
LIN {X 0.091,Y -650.125,Z 933.530,A 0.000,B 0.000,C 90.000,E1 131.434} C_DIS
LIN {X -0.078,Y -654.019,Z 933.525,A 0.000,B 0.000,C 90.000,E1 130.458} C_DIS
LIN {X 0.245,Y -661.482,Z 933.514,A 0.000,B 0.000,C 90.000,E1 128.463} C_DIS
LIN {X -0.123,Y -667.007,Z 933.506,A 0.000,B 0.000,C 90.000,E1 127.030} C_DIS
LIN {X 0.447,Y -670.610,Z 933.500,A 0.000,B 0.000,C 90.000,E1 126.011} C_DIS
LIN {X -0.271,Y -674.067,Z 933.495,A 0.000,B 0.000,C 90.000,E1 125.105} C_DIS
LIN {X 0.154,Y -678.028,Z 933.488,A 0.000,B 0.000,C 90.000,E1 123.865} C_DIS
LIN {X 0.095,Y -680.872,Z 933.483,A 0.000,B 0.000,C 90.000,E1 122.911} C_DIS
LIN {X -0.123,Y -682.853,Z 933.479,A 0.000,B 0.000,C 90.000,E1 122.212} C_DIS
LIN {X 0.252,Y -684.618,Z 933.475,A 0.000,B 0.000,C 90.000,E1 121.465} C_DIS
LIN {X 0.131,Y -687.262,Z 933.468,A 0.000,B 0.000,C 90.000,E1 120.285} C_DIS
LIN {X 0.398,Y -689.340,Z 933.462,A 0.000,B 0.000,C 90.000,E1 119.077} C_DIS
LIN {X 0.255,Y -690.151,Z 933.459,A 0.000,B 0.000,C 90.000,E1 118.615} C_DIS
LIN {X -0.345,Y -691.301,Z 933.454,A 0.000,B 0.000,C 90.000,E1 117.719} C_DIS
LIN {X 0.005,Y -692.064,Z 933.449,A 0.000,B 0.000,C 90.000,E1 116.744} C_DIS
LIN {X -0.130,Y -692.311,Z 933.446,A 0.000,B 0.000,C 90.000,E1 116.283} C_DIS
LIN {X 0.160,Y -692.501,Z 933.439,A 0.000,B 0.000,C 90.000,E1 115.079} C_DIS
LIN {X -0.032,Y -692.381,Z 933.436,A 0.000,B 0.000,C 90.000,E1 114.387} C_DIS
LIN {X 0.169,Y -692.182,Z 933.433,A 0.000,B 0.000,C 90.000,E1 113.898} C_DIS
LIN {X -0.262,Y -691.620,Z 933.430,A 0.000,B 0.000,C 90.000,E1 113.462} C_DIS
LIN {X -0.024,Y -691.010,Z 933.429,A 0.000,B 0.000,C 90.000,E1 113.206} C_DIS
LIN {X 0.212,Y -690.232,Z 933.428,A 0.000,B 0.000,C 90.000,E1 112.950} C_DIS
LIN {X 0.177,Y -689.304,Z 933.426,A 0.000,B 0.000,C 90.000,E1 112.717} C_DIS
LIN {X -0.343,Y -688.614,Z 933.426,A 0.000,B 0.000,C 90.000,E1 112.642} C_DIS
LIN {X -0.118,Y -686.418,Z 933.424,A 0.000,B 0.000,C 90.000,E1 112.386} C_DIS
LIN {X -0.155,Y -684.077,Z 933.423,A 0.000,B 0.000,C 90.000,E1 112.153} C_DIS
LIN {X -0.042,Y -682.689,Z 933.422,A 0.000,B 0.000,C 90.000,E1 112.025} C_DIS
LIN {X 0.165,Y -680.858,Z 933.422,A 0.000,B 0.000,C 90.000,E1 111.897} C_DIS
LIN {X 0.119,Y -678.124,Z 933.421,A 0.000,B 0.000,C 90.000,E1 111.791} C_DIS
LIN {X 0.205,Y -676.044,Z 933.421,A 0.000,B 0.000,C 90.000,E1 111.716} C_DIS
LIN {X 0.065,Y -667.912,Z 933.420,A 0.000,B 0.000,C 90.000,E1 111.535} C_DIS
LIN {X 0.120,Y -660.497,Z 933.419,A 0.000,B 0.000,C 90.000,E1 111.482} C_DIS
LIN {X 0.077,Y -640.219,Z 933.419,A 0.000,B 0.000,C 90.000,E1 111.482} C_DIS
LIN {X 0.251,Y -633.536,Z 933.419,A 0.000,B 0.000,C 90.000,E1 111.408} C_DIS
LIN {X -0.103,Y -627.796,Z 933.419,A 0.000,B 0.000,C 90.000,E1 111.354} C_DIS
LIN {X 0.034,Y -622.191,Z 933.418,A 0.000,B 0.000,C 90.000,E1 111.227} C_DIS
LIN {X -0.164,Y -615.210,Z 933.417,A 0.000,B 0.000,C 90.000,E1 111.046} C_DIS
LIN {X -0.200,Y -608.346,Z 933.415,A 0.000,B 0.000,C 90.000,E1 110.791} C_DIS
LIN {X 0.346,Y -602.659,Z 933.414,A 0.000,B 0.000,C 90.000,E1 110.482} C_DIS
LIN {X 0.236,Y -596.041,Z 933.412,A 0.000,B 0.000,C 90.000,E1 110.120} C_DIS
LIN {X -0.077,Y -589.045,Z 933.409,A 0.000,B 0.000,C 90.000,E1 109.685} C_DIS
LIN {X 0.065,Y -583.444,Z 933.407,A 0.000,B 0.000,C 90.000,E1 109.268} C_DIS
LIN {X 0.016,Y -578.943,Z 933.405,A 0.000,B 0.000,C 90.000,E1 108.960} C_DIS
LIN {X -0.081,Y -573.794,Z 933.404,A 0.000,B 0.000,C 90.000,E1 108.671} C_DIS
LIN {X -0.215,Y -568.640,Z 933.402,A 0.000,B 0.000,C 90.000,E1 108.417} C_DIS
LIN {X -0.300,Y -563.129,Z 933.401,A 0.000,B 0.000,C 90.000,E1 108.181} C_DIS
LIN {X 0.008,Y -556.687,Z 933.399,A 0.000,B 0.000,C 90.000,E1 107.873} C_DIS
LIN {X -0.099,Y -554.245,Z 933.399,A 0.000,B 0.000,C 90.000,E1 107.764} C_DIS
LIN {X 0.127,Y -552.498,Z 933.398,A 0.000,B 0.000,C 90.000,E1 107.583} C_DIS
LIN {X 0.091,Y -552.475,Z 933.398,A 0.000,B 0.000,C 90.000,E1 107.583} C_DIS
LIN {X 0.025,Y -552.049,Z 933.396,A 0.000,B 0.000,C 90.000,E1 107.330} C_DIS
LIN {X 0.317,Y -552.740,Z 933.386,A 0.000,B 0.000,C 90.000,E1 105.481} C_DIS
LIN {X 0.208,Y -553.649,Z 933.375,A 0.000,B 0.000,C 90.000,E1 103.536} C_DIS
LIN {X 0.121,Y -554.850,Z 933.365,A 0.000,B 0.000,C 90.000,E1 101.591} C_DIS
LIN {X -0.034,Y -556.639,Z 933.352,A 0.000,B 0.000,C 90.000,E1 99.378} C_DIS
LIN {X 0.049,Y -557.978,Z 933.343,A 0.000,B 0.000,C 90.000,E1 97.701} C_DIS
LIN {X -0.107,Y -558.767,Z 933.337,A 0.000,B 0.000,C 90.000,E1 96.606} C_DIS
LIN {X -0.117,Y -559.657,Z 933.329,A 0.000,B 0.000,C 90.000,E1 95.220} C_DIS
LIN {X -0.082,Y -560.592,Z 933.320,A 0.000,B 0.000,C 90.000,E1 93.555} C_DIS
LIN {X -0.246,Y -561.181,Z 933.314,A 0.000,B 0.000,C 90.000,E1 92.465} C_DIS
LIN {X -0.209,Y -561.906,Z 933.304,A 0.000,B 0.000,C 90.000,E1 90.802} C_DIS
LIN {X 0.191,Y -562.250,Z 933.298,A 0.000,B 0.000,C 90.000,E1 89.656} C_DIS
LIN {X 0.133,Y -562.618,Z 933.291,A 0.000,B 0.000,C 90.000,E1 88.282} C_DIS
LIN {X 0.223,Y -562.963,Z 933.281,A 0.000,B 0.000,C 90.000,E1 86.617} C_DIS
LIN {X -0.233,Y -563.246,Z 933.272,A 0.000,B 0.000,C 90.000,E1 85.008} C_DIS
LIN {X -0.224,Y -563.425,Z 933.265,A 0.000,B 0.000,C 90.000,E1 83.628} C_DIS
LIN {X -0.155,Y -563.661,Z 933.257,A 0.000,B 0.000,C 90.000,E1 82.243} C_DIS
LIN {X 0.165,Y -564.146,Z 933.248,A 0.000,B 0.000,C 90.000,E1 80.557} C_DIS
LIN {X 0.283,Y -565.040,Z 933.235,A 0.000,B 0.000,C 90.000,E1 78.342} C_DIS
LIN {X -0.019,Y -566.304,Z 933.223,A 0.000,B 0.000,C 90.000,E1 76.172} C_DIS
LIN {X 0.250,Y -567.010,Z 933.217,A 0.000,B 0.000,C 90.000,E1 75.046} C_DIS
LIN {X -0.069,Y -567.922,Z 933.208,A 0.000,B 0.000,C 90.000,E1 73.433} C_DIS
LIN {X 0.008,Y -568.686,Z 933.200,A 0.000,B 0.000,C 90.000,E1 72.054} C_DIS
LIN {X 0.046,Y -569.552,Z 933.190,A 0.000,B 0.000,C 90.000,E1 70.134} C_DIS
LIN {X 0.332,Y -570.090,Z 933.181,A 0.000,B 0.000,C 90.000,E1 68.465} C_DIS
LIN {X -0.284,Y -570.504,Z 933.170,A 0.000,B 0.000,C 90.000,E1 66.613} C_DIS
LIN {X 0.072,Y -570.714,Z 933.164,A 0.000,B 0.000,C 90.000,E1 65.485} C_DIS
LIN {X 0.088,Y -570.916,Z 933.155,A 0.000,B 0.000,C 90.000,E1 63.845} C_DIS
LIN {X -0.160,Y -570.999,Z 933.150,A 0.000,B 0.000,C 90.000,E1 63.050} C_DIS
LIN {X -0.054,Y -571.118,Z 933.144,A 0.000,B 0.000,C 90.000,E1 61.948} C_DIS
LIN {X -0.289,Y -571.076,Z 933.135,A 0.000,B 0.000,C 90.000,E1 60.333} C_DIS
LIN {X -0.084,Y -571.099,Z 933.128,A 0.000,B 0.000,C 90.000,E1 58.948} C_DIS
LIN {X -0.018,Y -570.995,Z 933.123,A 0.000,B 0.000,C 90.000,E1 58.122} C_DIS
LIN {X -0.057,Y -570.447,Z 933.112,A 0.000,B 0.000,C 90.000,E1 56.215} C_DIS
LIN {X 0.139,Y -569.838,Z 933.106,A 0.000,B 0.000,C 90.000,E1 55.102} C_DIS
LIN {X -0.008,Y -569.045,Z 933.099,A 0.000,B 0.000,C 90.000,E1 53.749} C_DIS
LIN {X 0.158,Y -568.107,Z 933.093,A 0.000,B 0.000,C 90.000,E1 52.637} C_DIS
LIN {X 0.077,Y -567.275,Z 933.088,A 0.000,B 0.000,C 90.000,E1 51.823} C_DIS
LIN {X 0.109,Y -565.920,Z 933.082,A 0.000,B 0.000,C 90.000,E1 50.723} C_DIS
LIN {X 0.115,Y -564.394,Z 933.076,A 0.000,B 0.000,C 90.000,E1 49.622} C_DIS
LIN {X -0.007,Y -563.010,Z 933.071,A 0.000,B 0.000,C 90.000,E1 48.809} C_DIS
LIN {X -0.104,Y -560.833,Z 933.065,A 0.000,B 0.000,C 90.000,E1 47.715} C_DIS
LIN {X 0.107,Y -558.957,Z 933.060,A 0.000,B 0.000,C 90.000,E1 46.863} C_DIS
LIN {X 0.339,Y -556.030,Z 933.054,A 0.000,B 0.000,C 90.000,E1 45.729} C_DIS
LIN {X 0.098,Y -553.483,Z 933.050,A 0.000,B 0.000,C 90.000,E1 44.919} C_DIS
LIN {X -0.170,Y -550.676,Z 933.045,A 0.000,B 0.000,C 90.000,E1 44.109} C_DIS
LIN {X -0.105,Y -548.602,Z 933.042,A 0.000,B 0.000,C 90.000,E1 43.542} C_DIS
LIN {X -0.027,Y -545.155,Z 933.037,A 0.000,B 0.000,C 90.000,E1 42.690} C_DIS
LIN {X -0.178,Y -542.011,Z 933.033,A 0.000,B 0.000,C 90.000,E1 42.000} C_DIS
LIN {X 0.218,Y -539.271,Z 933.030,A 0.000,B 0.000,C 90.000,E1 41.391} C_DIS
LIN {X -0.166,Y -536.323,Z 933.027,A 0.000,B 0.000,C 90.000,E1 40.862} C_DIS
LIN {X 0.184,Y -533.182,Z 933.024,A 0.000,B 0.000,C 90.000,E1 40.253} C_DIS
LIN {X -0.079,Y -528.914,Z 933.020,A 0.000,B 0.000,C 90.000,E1 39.564} C_DIS
LIN {X -0.008,Y -522.683,Z 933.014,A 0.000,B 0.000,C 90.000,E1 38.543} C_DIS
LIN {X 0.040,Y -517.919,Z 933.010,A 0.000,B 0.000,C 90.000,E1 37.810} C_DIS
LIN {X -0.033,Y -510.755,Z 933.004,A 0.000,B 0.000,C 90.000,E1 36.790} C_DIS
LIN {X 0.308,Y -505.222,Z 933.000,A 0.000,B 0.000,C 90.000,E1 36.011} C_DIS
LIN {X 0.014,Y -499.414,Z 932.996,A 0.000,B 0.000,C 90.000,E1 35.311} C_DIS
LIN {X -0.076,Y -494.403,Z 932.993,A 0.000,B 0.000,C 90.000,E1 34.739} C_DIS
LIN {X 0.210,Y -489.100,Z 932.990,A 0.000,B 0.000,C 90.000,E1 34.119} C_DIS
LIN {X -0.002,Y -482.023,Z 932.986,A 0.000,B 0.000,C 90.000,E1 33.420} C_DIS
LIN {X 0.293,Y -473.332,Z 932.981,A 0.000,B 0.000,C 90.000,E1 32.546} C_DIS
LIN {X -0.070,Y -464.637,Z 932.977,A 0.000,B 0.000,C 90.000,E1 31.799} C_DIS
LIN {X -0.022,Y -457.094,Z 932.973,A 0.000,B 0.000,C 90.000,E1 31.131} C_DIS
LIN {X 0.048,Y -446.319,Z 932.968,A 0.000,B 0.000,C 90.000,E1 30.207} C_DIS
LIN {X 0.245,Y -426.340,Z 932.958,A 0.000,B 0.000,C 90.000,E1 28.487} C_DIS
LIN {X 0.041,Y -409.753,Z 932.950,A 0.000,B 0.000,C 90.000,E1 27.001} C_DIS
LIN {X 0.136,Y -398.513,Z 932.944,A 0.000,B 0.000,C 90.000,E1 25.848} C_DIS
LIN {X 0.091,Y -396.326,Z 932.942,A 0.000,B 0.000,C 90.000,E1 25.591} C_DIS
LIN {X -0.101,Y -392.648,Z 932.939,A 0.000,B 0.000,C 90.000,E1 25.079} C_DIS
LIN {X 0.135,Y -390.269,Z 932.936,A 0.000,B 0.000,C 90.000,E1 24.515} C_DIS
LIN {X 0.067,Y -389.303,Z 932.934,A 0.000,B 0.000,C 90.000,E1 24.079} C_DIS
LIN {X -0.075,Y -388.901,Z 932.930,A 0.000,B 0.000,C 90.000,E1 23.387} C_DIS
LIN {X -0.116,Y -389.210,Z 932.924,A 0.000,B 0.000,C 90.000,E1 22.333} C_DIS
LIN {X -0.167,Y -392.510,Z 932.904,A 0.000,B 0.000,C 90.000,E1 18.779} C_DIS
LIN {X 0.097,Y -395.364,Z 932.890,A 0.000,B 0.000,C 90.000,E1 16.260} C_DIS
LIN {X -0.086,Y -399.003,Z 932.875,A 0.000,B 0.000,C 90.000,E1 13.467} C_DIS
LIN {X -0.043,Y -403.157,Z 932.859,A 0.000,B 0.000,C 90.000,E1 10.658} C_DIS
LIN {X -0.036,Y -406.000,Z 932.850,A 0.000,B 0.000,C 90.000,E1 8.916} C_DIS
LIN {X 0.009,Y -410.281,Z 932.836,A 0.000,B 0.000,C 90.000,E1 6.486} C_DIS
LIN {X 0.083,Y -415.619,Z 932.821,A 0.000,B 0.000,C 90.000,E1 3.726} C_DIS
LIN {X -0.096,Y -422.367,Z 932.804,A 0.000,B 0.000,C 90.000,E1 0.688} C_DIS
LIN {X -0.108,Y -427.031,Z 932.793,A 0.000,B 0.000,C 90.000,E1 358.797} C_DIS
LIN {X 0.024,Y -429.062,Z 932.790,A 0.000,B 0.000,C 90.000,E1 358.108} C_DIS
LIN {X 0.180,Y -431.112,Z 932.787,A 0.000,B 0.000,C 90.000,E1 357.593} C_DIS
LIN {X 0.104,Y -434.068,Z 932.784,A 0.000,B 0.000,C 90.000,E1 357.135} C_DIS
LIN {X 0.144,Y -435.336,Z 932.783,A 0.000,B 0.000,C 90.000,E1 356.963} C_DIS
LIN {X 0.209,Y -437.044,Z 932.782,A 0.000,B 0.000,C 90.000,E1 356.788} C_DIS
LIN {X 0.148,Y -441.441,Z 932.780,A 0.000,B 0.000,C 90.000,E1 356.445} C_DIS
LIN {X 0.168,Y -449.611,Z 932.778,A 0.000,B 0.000,C 90.000,E1 356.045} C_DIS
LIN {X -0.041,Y -459.850,Z 932.776,A 0.000,B 0.000,C 90.000,E1 355.584} C_DIS
LIN {X 0.039,Y -466.492,Z 932.774,A 0.000,B 0.000,C 90.000,E1 355.241} C_DIS
LIN {X -0.182,Y -481.566,Z 932.769,A 0.000,B 0.000,C 90.000,E1 354.489} C_DIS
LIN {X -0.010,Y -489.929,Z 932.767,A 0.000,B 0.000,C 90.000,E1 354.033} C_DIS
LIN {X 0.214,Y -499.892,Z 932.764,A 0.000,B 0.000,C 90.000,E1 353.457} C_DIS
LIN {X -0.114,Y -509.535,Z 932.761,A 0.000,B 0.000,C 90.000,E1 352.932} C_DIS
LIN {X 0.221,Y -519.001,Z 932.757,A 0.000,B 0.000,C 90.000,E1 352.299} C_DIS
LIN {X 0.180,Y -525.210,Z 932.755,A 0.000,B 0.000,C 90.000,E1 351.894} C_DIS
LIN {X 0.034,Y -529.469,Z 932.753,A 0.000,B 0.000,C 90.000,E1 351.602} C_DIS
LIN {X 0.153,Y -535.383,Z 932.751,A 0.000,B 0.000,C 90.000,E1 351.141} C_DIS
LIN {X 0.114,Y -542.528,Z 932.748,A 0.000,B 0.000,C 90.000,E1 350.557} C_DIS
LIN {X 0.207,Y -549.331,Z 932.744,A 0.000,B 0.000,C 90.000,E1 349.926} C_DIS
LIN {X -0.242,Y -554.571,Z 932.741,A 0.000,B 0.000,C 90.000,E1 349.454} C_DIS
LIN {X 0.156,Y -559.594,Z 932.738,A 0.000,B 0.000,C 90.000,E1 348.870} C_DIS
LIN {X -0.189,Y -567.567,Z 932.733,A 0.000,B 0.000,C 90.000,E1 347.937} C_DIS
LIN {X -0.143,Y -570.757,Z 932.731,A 0.000,B 0.000,C 90.000,E1 347.521} C_DIS
LIN {X 0.238,Y -574.742,Z 932.728,A 0.000,B 0.000,C 90.000,E1 346.937} C_DIS
LIN {X -0.263,Y -580.472,Z 932.723,A 0.000,B 0.000,C 90.000,E1 346.172} C_DIS
LIN {X 0.238,Y -587.205,Z 932.717,A 0.000,B 0.000,C 90.000,E1 345.046} C_DIS
LIN {X -0.227,Y -592.658,Z 932.712,A 0.000,B 0.000,C 90.000,E1 344.157} C_DIS
LIN {X -0.035,Y -594.867,Z 932.710,A 0.000,B 0.000,C 90.000,E1 343.740} C_DIS
LIN {X 0.094,Y -600.342,Z 932.704,A 0.000,B 0.000,C 90.000,E1 342.670} C_DIS
LIN {X 0.123,Y -608.039,Z 932.695,A 0.000,B 0.000,C 90.000,E1 341.094} C_DIS
LIN {X 0.016,Y -613.431,Z 932.689,A 0.000,B 0.000,C 90.000,E1 339.934} C_DIS
LIN {X -0.003,Y -617.868,Z 932.683,A 0.000,B 0.000,C 90.000,E1 338.901} C_DIS
LIN {X 0.260,Y -622.018,Z 932.677,A 0.000,B 0.000,C 90.000,E1 337.847} C_DIS
LIN {X 0.006,Y -625.014,Z 932.673,A 0.000,B 0.000,C 90.000,E1 337.102} C_DIS
LIN {X -0.221,Y -627.824,Z 932.669,A 0.000,B 0.000,C 90.000,E1 336.357} C_DIS
LIN {X 0.199,Y -632.203,Z 932.662,A 0.000,B 0.000,C 90.000,E1 335.049} C_DIS
LIN {X 0.343,Y -635.498,Z 932.656,A 0.000,B 0.000,C 90.000,E1 334.024} C_DIS
LIN {X 0.025,Y -639.269,Z 932.649,A 0.000,B 0.000,C 90.000,E1 332.794} C_DIS
LIN {X 0.335,Y -642.750,Z 932.642,A 0.000,B 0.000,C 90.000,E1 331.513} C_DIS
LIN {X 0.051,Y -645.193,Z 932.636,A 0.000,B 0.000,C 90.000,E1 330.539} C_DIS
LIN {X 0.194,Y -648.180,Z 932.630,A 0.000,B 0.000,C 90.000,E1 329.282} C_DIS
LIN {X -0.256,Y -650.287,Z 932.624,A 0.000,B 0.000,C 90.000,E1 328.329} C_DIS
LIN {X -0.125,Y -652.082,Z 932.618,A 0.000,B 0.000,C 90.000,E1 327.327} C_DIS
LIN {X -0.064,Y -653.374,Z 932.614,A 0.000,B 0.000,C 90.000,E1 326.580} C_DIS
LIN {X -0.083,Y -654.823,Z 932.609,A 0.000,B 0.000,C 90.000,E1 325.595} C_DIS
LIN {X 0.004,Y -656.364,Z 932.602,A 0.000,B 0.000,C 90.000,E1 324.356} C_DIS
LIN {X -0.091,Y -657.938,Z 932.594,A 0.000,B 0.000,C 90.000,E1 322.889} C_DIS
LIN {X -0.093,Y -658.946,Z 932.587,A 0.000,B 0.000,C 90.000,E1 321.662} C_DIS
LIN {X 0.353,Y -660.317,Z 932.578,A 0.000,B 0.000,C 90.000,E1 319.908} C_DIS
LIN {X -0.210,Y -661.938,Z 932.567,A 0.000,B 0.000,C 90.000,E1 318.000} C_DIS
LIN {X 0.228,Y -662.590,Z 932.563,A 0.000,B 0.000,C 90.000,E1 317.229} C_DIS
LIN {X -0.300,Y -663.820,Z 932.554,A 0.000,B 0.000,C 90.000,E1 315.810} C_DIS
LIN {X 0.117,Y -666.088,Z 932.540,A 0.000,B 0.000,C 90.000,E1 313.095} C_DIS
LIN {X -0.347,Y -667.463,Z 932.531,A 0.000,B 0.000,C 90.000,E1 311.676} C_DIS
LIN {X 0.211,Y -668.823,Z 932.523,A 0.000,B 0.000,C 90.000,E1 310.172} C_DIS
LIN {X 0.285,Y -669.686,Z 932.518,A 0.000,B 0.000,C 90.000,E1 309.197} C_DIS
LIN {X -0.052,Y -670.471,Z 932.513,A 0.000,B 0.000,C 90.000,E1 308.257} C_DIS
LIN {X 0.031,Y -671.195,Z 932.507,A 0.000,B 0.000,C 90.000,E1 307.282} C_DIS
LIN {X 0.248,Y -671.725,Z 932.502,A 0.000,B 0.000,C 90.000,E1 306.297} C_DIS
LIN {X 0.296,Y -672.456,Z 932.490,A 0.000,B 0.000,C 90.000,E1 304.119} C_DIS
LIN {X 0.022,Y -673.365,Z 932.479,A 0.000,B 0.000,C 90.000,E1 302.212} C_DIS
LIN {X -0.068,Y -674.764,Z 932.467,A 0.000,B 0.000,C 90.000,E1 300.050} C_DIS
LIN {X 0.215,Y -680.709,Z 932.442,A 0.000,B 0.000,C 90.000,E1 295.463} C_DIS
LIN {X 0.324,Y -682.527,Z 932.435,A 0.000,B 0.000,C 90.000,E1 294.259} C_DIS
LIN {X 0.039,Y -683.442,Z 932.431,A 0.000,B 0.000,C 90.000,E1 293.567} C_DIS
LIN {X 0.182,Y -683.953,Z 932.428,A 0.000,B 0.000,C 90.000,E1 293.078} C_DIS
LIN {X -0.299,Y -684.125,Z 932.426,A 0.000,B 0.000,C 90.000,E1 292.642} C_DIS
LIN {X -0.092,Y -684.021,Z 932.424,A 0.000,B 0.000,C 90.000,E1 292.386} C_DIS
LIN {X 0.061,Y -683.316,Z 932.422,A 0.000,B 0.000,C 90.000,E1 291.897} C_DIS
LIN {X 0.010,Y -682.509,Z 932.420,A 0.000,B 0.000,C 90.000,E1 291.663} C_DIS
LIN {X 0.111,Y -681.699,Z 932.420,A 0.000,B 0.000,C 90.000,E1 291.535} C_DIS
LIN {X 0.157,Y -678.520,Z 932.418,A 0.000,B 0.000,C 90.000,E1 291.173} C_DIS
LIN {X 0.250,Y -677.508,Z 932.417,A 0.000,B 0.000,C 90.000,E1 291.046} C_DIS
LIN {X -0.290,Y -676.094,Z 932.416,A 0.000,B 0.000,C 90.000,E1 290.972} C_DIS
LIN {X -0.134,Y -669.433,Z 932.414,A 0.000,B 0.000,C 90.000,E1 290.556} C_DIS
LIN {X -0.258,Y -664.865,Z 932.413,A 0.000,B 0.000,C 90.000,E1 290.301} C_DIS
LIN {X 0.193,Y -663.542,Z 932.412,A 0.000,B 0.000,C 90.000,E1 290.174} C_DIS
LIN {X 0.020,Y -662.129,Z 932.412,A 0.000,B 0.000,C 90.000,E1 290.066} C_DIS
LIN {X -0.020,Y -662.110,Z 932.411,A 0.000,B 0.000,C 90.000,E1 290.066} C_DIS
LIN {X -0.126,Y -661.846,Z 932.411,A 0.000,B 0.000,C 90.000,E1 289.939} C_DIS
LIN {X -0.087,Y -662.411,Z 932.409,A 0.000,B 0.000,C 90.000,E1 289.577} C_DIS
LIN {X -0.074,Y -664.206,Z 932.406,A 0.000,B 0.000,C 90.000,E1 289.087} C_DIS
LIN {X -0.043,Y -671.608,Z 932.398,A 0.000,B 0.000,C 90.000,E1 287.638} C_DIS
LIN {X 0.018,Y -673.962,Z 932.395,A 0.000,B 0.000,C 90.000,E1 287.149} C_DIS
LIN {X -0.160,Y -677.009,Z 932.391,A 0.000,B 0.000,C 90.000,E1 286.441} C_DIS
LIN {X -0.119,Y -679.432,Z 932.387,A 0.000,B 0.000,C 90.000,E1 285.717} C_DIS
LIN {X -0.202,Y -680.763,Z 932.385,A 0.000,B 0.000,C 90.000,E1 285.245} C_DIS
LIN {X -0.339,Y -682.943,Z 932.379,A 0.000,B 0.000,C 90.000,E1 284.300} C_DIS
LIN {X 0.269,Y -683.879,Z 932.377,A 0.000,B 0.000,C 90.000,E1 283.772} C_DIS
LIN {X 0.175,Y -685.433,Z 932.371,A 0.000,B 0.000,C 90.000,E1 282.827} C_DIS
LIN {X 0.113,Y -686.338,Z 932.367,A 0.000,B 0.000,C 90.000,E1 282.119} C_DIS
LIN {X -0.067,Y -686.786,Z 932.365,A 0.000,B 0.000,C 90.000,E1 281.658} C_DIS
LIN {X -0.103,Y -687.039,Z 932.362,A 0.000,B 0.000,C 90.000,E1 281.186} C_DIS
LIN {X -0.141,Y -687.006,Z 932.359,A 0.000,B 0.000,C 90.000,E1 280.715} C_DIS
LIN {X -0.306,Y -686.627,Z 932.357,A 0.000,B 0.000,C 90.000,E1 280.254} C_DIS
LIN {X 0.348,Y -686.323,Z 932.356,A 0.000,B 0.000,C 90.000,E1 279.962} C_DIS
LIN {X 0.183,Y -685.404,Z 932.353,A 0.000,B 0.000,C 90.000,E1 279.500} C_DIS
LIN {X 0.125,Y -683.998,Z 932.350,A 0.000,B 0.000,C 90.000,E1 279.029} C_DIS
LIN {X -0.050,Y -682.218,Z 932.348,A 0.000,B 0.000,C 90.000,E1 278.568} C_DIS
LIN {X -0.232,Y -680.065,Z 932.345,A 0.000,B 0.000,C 90.000,E1 278.106} C_DIS
LIN {X 0.113,Y -675.874,Z 932.340,A 0.000,B 0.000,C 90.000,E1 277.239} C_DIS
LIN {X -0.267,Y -671.410,Z 932.336,A 0.000,B 0.000,C 90.000,E1 276.429} C_DIS
LIN {X 0.062,Y -667.797,Z 932.332,A 0.000,B 0.000,C 90.000,E1 275.796} C_DIS
LIN {X -0.213,Y -664.472,Z 932.330,A 0.000,B 0.000,C 90.000,E1 275.334} C_DIS
LIN {X 0.057,Y -659.721,Z 932.326,A 0.000,B 0.000,C 90.000,E1 274.702} C_DIS
LIN {X -0.321,Y -655.591,Z 932.323,A 0.000,B 0.000,C 90.000,E1 274.245} C_DIS
LIN {X -0.126,Y -649.885,Z 932.320,A 0.000,B 0.000,C 90.000,E1 273.612} C_DIS
LIN {X 0.222,Y -645.026,Z 932.317,A 0.000,B 0.000,C 90.000,E1 273.094} C_DIS
LIN {X 0.053,Y -638.463,Z 932.314,A 0.000,B 0.000,C 90.000,E1 272.522} C_DIS
LIN {X 0.220,Y -631.469,Z 932.311,A 0.000,B 0.000,C 90.000,E1 271.949} C_DIS
LIN {X 0.161,Y -624.033,Z 932.308,A 0.000,B 0.000,C 90.000,E1 271.432} C_DIS
LIN {X 0.183,Y -617.870,Z 932.306,A 0.000,B 0.000,C 90.000,E1 271.031} C_DIS
LIN {X -0.170,Y -611.578,Z 932.304,A 0.000,B 0.000,C 90.000,E1 270.688} C_DIS
LIN {X 0.104,Y -603.429,Z 932.301,A 0.000,B 0.000,C 90.000,E1 270.229} C_DIS
LIN {X -0.278,Y -596.576,Z 932.300,A 0.000,B 0.000,C 90.000,E1 269.943} C_DIS
LIN {X -0.220,Y -591.340,Z 932.298,A 0.000,B 0.000,C 90.000,E1 269.714} C_DIS
LIN {X -0.025,Y -583.883,Z 932.297,A 0.000,B 0.000,C 90.000,E1 269.427} C_DIS
LIN {X -0.008,Y -578.091,Z 932.296,A 0.000,B 0.000,C 90.000,E1 269.255} C_DIS
LIN {X -0.107,Y -570.268,Z 932.295,A 0.000,B 0.000,C 90.000,E1 269.083} C_DIS
LIN {X -0.036,Y -564.592,Z 932.294,A 0.000,B 0.000,C 90.000,E1 268.969} C_DIS
LIN {X -0.153,Y -557.796,Z 932.294,A 0.000,B 0.000,C 90.000,E1 268.912} C_DIS
LIN {X -0.005,Y -552.050,Z 932.294,A 0.000,B 0.000,C 90.000,E1 268.854} C_DIS
LIN {X -0.222,Y -550.971,Z 932.294,A 0.000,B 0.000,C 90.000,E1 268.854} C_DIS
LIN {X -0.268,Y -550.768,Z 932.294,A 0.000,B 0.000,C 90.000,E1 268.854} C_DIS
LIN {X -0.095,Y -549.282,Z 932.292,A 0.000,B 0.000,C 90.000,E1 268.625} C_DIS
LIN {X 0.256,Y -545.631,Z 932.290,A 0.000,B 0.000,C 90.000,E1 268.167} C_DIS
LIN {X 0.066,Y -544.111,Z 932.289,A 0.000,B 0.000,C 90.000,E1 268.051} C_DIS
LIN {X 0.024,Y -544.079,Z 932.289,A 0.000,B 0.000,C 90.000,E1 268.051} C_DIS
LIN {X 0.062,Y -543.395,Z 932.288,A 0.000,B 0.000,C 90.000,E1 267.764} C_DIS
LIN {X 0.204,Y -540.219,Z 932.268,A 0.000,B 0.000,C 90.000,E1 264.204} C_DIS
LIN {X -0.072,Y -539.107,Z 932.258,A 0.000,B 0.000,C 90.000,E1 262.527} C_DIS
LIN {X 0.102,Y -538.104,Z 932.251,A 0.000,B 0.000,C 90.000,E1 261.084} C_DIS
LIN {X 0.205,Y -537.345,Z 932.246,A 0.000,B 0.000,C 90.000,E1 260.218} C_DIS
LIN {X -0.138,Y -536.296,Z 932.241,A 0.000,B 0.000,C 90.000,E1 259.398} C_DIS
LIN {X 0.148,Y -534.202,Z 932.233,A 0.000,B 0.000,C 90.000,E1 257.937} C_DIS
LIN {X 0.081,Y -531.663,Z 932.222,A 0.000,B 0.000,C 90.000,E1 255.936} C_DIS
LIN {X -0.152,Y -530.311,Z 932.216,A 0.000,B 0.000,C 90.000,E1 254.810} C_DIS
LIN {X -0.233,Y -528.589,Z 932.208,A 0.000,B 0.000,C 90.000,E1 253.378} C_DIS
LIN {X 0.151,Y -526.800,Z 932.200,A 0.000,B 0.000,C 90.000,E1 251.891} C_DIS
LIN {X -0.177,Y -524.569,Z 932.190,A 0.000,B 0.000,C 90.000,E1 250.188} C_DIS
LIN {X -0.036,Y -522.715,Z 932.182,A 0.000,B 0.000,C 90.000,E1 248.720} C_DIS
LIN {X 0.263,Y -520.812,Z 932.174,A 0.000,B 0.000,C 90.000,E1 247.230} C_DIS
LIN {X 0.049,Y -518.607,Z 932.166,A 0.000,B 0.000,C 90.000,E1 245.793} C_DIS
LIN {X 0.012,Y -516.337,Z 932.157,A 0.000,B 0.000,C 90.000,E1 244.332} C_DIS
LIN {X -0.075,Y -515.001,Z 932.153,A 0.000,B 0.000,C 90.000,E1 243.461} C_DIS
LIN {X -0.062,Y -513.046,Z 932.146,A 0.000,B 0.000,C 90.000,E1 242.281} C_DIS
LIN {X 0.025,Y -510.573,Z 932.138,A 0.000,B 0.000,C 90.000,E1 240.795} C_DIS
LIN {X -0.024,Y -508.507,Z 932.131,A 0.000,B 0.000,C 90.000,E1 239.616} C_DIS
LIN {X 0.151,Y -506.352,Z 932.125,A 0.000,B 0.000,C 90.000,E1 238.408} C_DIS
LIN {X -0.133,Y -503.873,Z 932.118,A 0.000,B 0.000,C 90.000,E1 237.248} C_DIS
LIN {X 0.128,Y -500.489,Z 932.110,A 0.000,B 0.000,C 90.000,E1 235.722} C_DIS
LIN {X -0.078,Y -495.015,Z 932.096,A 0.000,B 0.000,C 90.000,E1 233.336} C_DIS
LIN {X -0.096,Y -491.784,Z 932.088,A 0.000,B 0.000,C 90.000,E1 231.823} C_DIS
LIN {X 0.127,Y -488.389,Z 932.079,A 0.000,B 0.000,C 90.000,E1 230.275} C_DIS
LIN {X 0.052,Y -484.224,Z 932.069,A 0.000,B 0.000,C 90.000,E1 228.447} C_DIS
LIN {X -0.123,Y -480.003,Z 932.059,A 0.000,B 0.000,C 90.000,E1 226.620} C_DIS
LIN {X -0.085,Y -475.955,Z 932.049,A 0.000,B 0.000,C 90.000,E1 224.757} C_DIS
LIN {X 0.108,Y -472.526,Z 932.040,A 0.000,B 0.000,C 90.000,E1 223.176} C_DIS
LIN {X -0.007,Y -468.340,Z 932.030,A 0.000,B 0.000,C 90.000,E1 221.310} C_DIS
LIN {X 0.035,Y -462.210,Z 932.014,A 0.000,B 0.000,C 90.000,E1 218.463} C_DIS
LIN {X 0.060,Y -458.783,Z 932.005,A 0.000,B 0.000,C 90.000,E1 216.870} C_DIS
LIN {X -0.254,Y -455.331,Z 931.996,A 0.000,B 0.000,C 90.000,E1 215.311} C_DIS
LIN {X 0.113,Y -451.793,Z 931.987,A 0.000,B 0.000,C 90.000,E1 213.658} C_DIS
LIN {X -0.058,Y -446.794,Z 931.975,A 0.000,B 0.000,C 90.000,E1 211.416} C_DIS
LIN {X -0.050,Y -442.446,Z 931.964,A 0.000,B 0.000,C 90.000,E1 209.461} C_DIS
LIN {X -0.072,Y -439.678,Z 931.956,A 0.000,B 0.000,C 90.000,E1 208.153} C_DIS
LIN {X 0.051,Y -436.857,Z 931.949,A 0.000,B 0.000,C 90.000,E1 206.821} C_DIS
LIN {X 0.148,Y -433.177,Z 931.940,A 0.000,B 0.000,C 90.000,E1 205.155} C_DIS
LIN {X 0.164,Y -428.083,Z 931.927,A 0.000,B 0.000,C 90.000,E1 202.823} C_DIS
LIN {X 0.117,Y -424.355,Z 931.918,A 0.000,B 0.000,C 90.000,E1 201.153} C_DIS
LIN {X -0.156,Y -420.689,Z 931.908,A 0.000,B 0.000,C 90.000,E1 199.504} C_DIS
LIN {X 0.081,Y -415.998,Z 931.895,A 0.000,B 0.000,C 90.000,E1 197.094} C_DIS
LIN {X 0.159,Y -413.266,Z 931.888,A 0.000,B 0.000,C 90.000,E1 195.717} C_DIS
LIN {X 0.103,Y -409.723,Z 931.878,A 0.000,B 0.000,C 90.000,E1 194.008} C_DIS
LIN {X 0.089,Y -404.888,Z 931.865,A 0.000,B 0.000,C 90.000,E1 191.591} C_DIS
LIN {X 0.104,Y -401.501,Z 931.855,A 0.000,B 0.000,C 90.000,E1 189.849} C_DIS
LIN {X 0.035,Y -397.430,Z 931.843,A 0.000,B 0.000,C 90.000,E1 187.757} C_DIS
LIN {X -0.159,Y -393.996,Z 931.833,A 0.000,B 0.000,C 90.000,E1 186.024} C_DIS
LIN {X -0.024,Y -388.132,Z 931.816,A 0.000,B 0.000,C 90.000,E1 182.808} C_DIS
LIN {X -0.143,Y -382.989,Z 931.798,A 0.000,B 0.000,C 90.000,E1 179.599} C_DIS
LIN {X -0.099,Y -381.730,Z 931.792,A 0.000,B 0.000,C 90.000,E1 178.511} C_DIS
LIN {X 0.060,Y -381.131,Z 931.788,A 0.000,B 0.000,C 90.000,E1 177.764} C_DIS
LIN {X -0.182,Y -380.976,Z 931.784,A 0.000,B 0.000,C 90.000,E1 177.078} C_DIS
LIN {X -0.028,Y -381.139,Z 931.780,A 0.000,B 0.000,C 90.000,E1 176.331} C_DIS
LIN {X -0.154,Y -381.743,Z 931.778,A 0.000,B 0.000,C 90.000,E1 175.988} C_DIS
LIN {X 0.181,Y -382.165,Z 931.776,A 0.000,B 0.000,C 90.000,E1 175.584} C_DIS
LIN {X 0.056,Y -382.843,Z 931.774,A 0.000,B 0.000,C 90.000,E1 175.241} C_DIS
LIN {X 0.011,Y -384.042,Z 931.772,A 0.000,B 0.000,C 90.000,E1 174.894} C_DIS
LIN {X -0.049,Y -384.749,Z 931.771,A 0.000,B 0.000,C 90.000,E1 174.723} C_DIS
LIN {X 0.035,Y -386.984,Z 931.768,A 0.000,B 0.000,C 90.000,E1 174.318} C_DIS
LIN {X -0.040,Y -389.197,Z 931.767,A 0.000,B 0.000,C 90.000,E1 173.970} C_DIS
LIN {X 0.072,Y -395.350,Z 931.763,A 0.000,B 0.000,C 90.000,E1 173.280} C_DIS
LIN {X 0.008,Y -402.078,Z 931.760,A 0.000,B 0.000,C 90.000,E1 172.704} C_DIS
LIN {X -0.132,Y -413.137,Z 931.755,A 0.000,B 0.000,C 90.000,E1 171.894} C_DIS
LIN {X 0.111,Y -428.591,Z 931.748,A 0.000,B 0.000,C 90.000,E1 170.679} C_DIS
LIN {X -0.190,Y -436.389,Z 931.745,A 0.000,B 0.000,C 90.000,E1 170.095} C_DIS
LIN {X 0.013,Y -445.271,Z 931.741,A 0.000,B 0.000,C 90.000,E1 169.285} C_DIS
LIN {X 0.033,Y -454.230,Z 931.736,A 0.000,B 0.000,C 90.000,E1 168.465} C_DIS
LIN {X 0.070,Y -458.595,Z 931.734,A 0.000,B 0.000,C 90.000,E1 168.049} C_DIS
LIN {X -0.078,Y -465.618,Z 931.730,A 0.000,B 0.000,C 90.000,E1 167.353} C_DIS
LIN {X 0.065,Y -475.162,Z 931.724,A 0.000,B 0.000,C 90.000,E1 166.297} C_DIS
LIN {X 0.232,Y -481.561,Z 931.720,A 0.000,B 0.000,C 90.000,E1 165.519} C_DIS
LIN {X 0.135,Y -490.435,Z 931.714,A 0.000,B 0.000,C 90.000,E1 164.464} C_DIS
LIN {X 0.040,Y -495.165,Z 931.710,A 0.000,B 0.000,C 90.000,E1 163.866} C_DIS
LIN {X -0.036,Y -503.837,Z 931.704,A 0.000,B 0.000,C 90.000,E1 162.670} C_DIS
LIN {X -0.254,Y -516.058,Z 931.694,A 0.000,B 0.000,C 90.000,E1 160.913} C_DIS
LIN {X -0.027,Y -521.821,Z 931.689,A 0.000,B 0.000,C 90.000,E1 160.007} C_DIS
LIN {X 0.121,Y -531.143,Z 931.681,A 0.000,B 0.000,C 90.000,E1 158.539} C_DIS
LIN {X 0.070,Y -537.372,Z 931.675,A 0.000,B 0.000,C 90.000,E1 157.539} C_DIS
LIN {X -0.037,Y -547.732,Z 931.666,A 0.000,B 0.000,C 90.000,E1 155.845} C_DIS
LIN {X -0.139,Y -551.785,Z 931.662,A 0.000,B 0.000,C 90.000,E1 155.153} C_DIS
LIN {X -0.141,Y -558.842,Z 931.655,A 0.000,B 0.000,C 90.000,E1 153.896} C_DIS
LIN {X -0.195,Y -564.581,Z 931.649,A 0.000,B 0.000,C 90.000,E1 152.794} C_DIS
LIN {X -0.254,Y -568.716,Z 931.644,A 0.000,B 0.000,C 90.000,E1 151.975} C_DIS
LIN {X 0.024,Y -574.482,Z 931.637,A 0.000,B 0.000,C 90.000,E1 150.717} C_DIS
LIN {X -0.218,Y -576.395,Z 931.635,A 0.000,B 0.000,C 90.000,E1 150.333} C_DIS
LIN {X 0.253,Y -581.081,Z 931.629,A 0.000,B 0.000,C 90.000,E1 149.203} C_DIS
LIN {X 0.294,Y -585.539,Z 931.623,A 0.000,B 0.000,C 90.000,E1 148.122} C_DIS
LIN {X -0.096,Y -589.791,Z 931.617,A 0.000,B 0.000,C 90.000,E1 147.089} C_DIS
LIN {X -0.055,Y -595.007,Z 931.610,A 0.000,B 0.000,C 90.000,E1 145.754} C_DIS
LIN {X -0.103,Y -597.105,Z 931.607,A 0.000,B 0.000,C 90.000,E1 145.229} C_DIS
LIN {X -0.102,Y -601.946,Z 931.599,A 0.000,B 0.000,C 90.000,E1 143.909} C_DIS
LIN {X -0.253,Y -607.582,Z 931.591,A 0.000,B 0.000,C 90.000,E1 142.351} C_DIS
LIN {X -0.294,Y -615.303,Z 931.579,A 0.000,B 0.000,C 90.000,E1 140.275} C_DIS
LIN {X 0.275,Y -620.211,Z 931.572,A 0.000,B 0.000,C 90.000,E1 138.933} C_DIS
LIN {X 0.265,Y -630.142,Z 931.558,A 0.000,B 0.000,C 90.000,E1 136.377} C_DIS
LIN {X -0.195,Y -634.219,Z 931.552,A 0.000,B 0.000,C 90.000,E1 135.405} C_DIS
LIN {X 0.113,Y -640.012,Z 931.544,A 0.000,B 0.000,C 90.000,E1 133.866} C_DIS
LIN {X 0.243,Y -643.941,Z 931.538,A 0.000,B 0.000,C 90.000,E1 132.852} C_DIS
LIN {X -0.134,Y -649.715,Z 931.530,A 0.000,B 0.000,C 90.000,E1 131.391} C_DIS
LIN {X 0.122,Y -653.653,Z 931.524,A 0.000,B 0.000,C 90.000,E1 130.378} C_DIS
LIN {X 0.024,Y -661.126,Z 931.513,A 0.000,B 0.000,C 90.000,E1 128.418} C_DIS
LIN {X 0.057,Y -666.663,Z 931.505,A 0.000,B 0.000,C 90.000,E1 126.950} C_DIS
LIN {X -0.315,Y -670.273,Z 931.500,A 0.000,B 0.000,C 90.000,E1 126.011} C_DIS
LIN {X -0.103,Y -673.717,Z 931.495,A 0.000,B 0.000,C 90.000,E1 125.025} C_DIS
LIN {X 0.152,Y -676.904,Z 931.489,A 0.000,B 0.000,C 90.000,E1 124.040} C_DIS
LIN {X 0.248,Y -680.539,Z 931.483,A 0.000,B 0.000,C 90.000,E1 122.832} C_DIS
LIN {X 0.219,Y -683.082,Z 931.477,A 0.000,B 0.000,C 90.000,E1 121.878} C_DIS
LIN {X 0.216,Y -685.294,Z 931.472,A 0.000,B 0.000,C 90.000,E1 120.924} C_DIS
LIN {X 0.262,Y -686.861,Z 931.468,A 0.000,B 0.000,C 90.000,E1 120.207} C_DIS
LIN {X 0.182,Y -688.904,Z 931.461,A 0.000,B 0.000,C 90.000,E1 119.027} C_DIS
LIN {X 0.039,Y -689.721,Z 931.459,A 0.000,B 0.000,C 90.000,E1 118.565} C_DIS
LIN {X -0.240,Y -690.844,Z 931.453,A 0.000,B 0.000,C 90.000,E1 117.641} C_DIS
LIN {X 0.098,Y -691.580,Z 931.448,A 0.000,B 0.000,C 90.000,E1 116.668} C_DIS
LIN {X -0.106,Y -691.811,Z 931.444,A 0.000,B 0.000,C 90.000,E1 115.976} C_DIS
LIN {X -0.061,Y -691.952,Z 931.439,A 0.000,B 0.000,C 90.000,E1 115.027} C_DIS
LIN {X 0.421,Y -691.931,Z 931.436,A 0.000,B 0.000,C 90.000,E1 114.515} C_DIS
LIN {X 0.225,Y -691.485,Z 931.432,A 0.000,B 0.000,C 90.000,E1 113.823} C_DIS
LIN {X -0.211,Y -690.951,Z 931.430,A 0.000,B 0.000,C 90.000,E1 113.387} C_DIS
LIN {X -0.015,Y -689.427,Z 931.427,A 0.000,B 0.000,C 90.000,E1 112.898} C_DIS
LIN {X 0.215,Y -688.418,Z 931.426,A 0.000,B 0.000,C 90.000,E1 112.642} C_DIS
LIN {X 0.328,Y -687.552,Z 931.425,A 0.000,B 0.000,C 90.000,E1 112.514} C_DIS
LIN {X -0.238,Y -684.193,Z 931.423,A 0.000,B 0.000,C 90.000,E1 112.206} C_DIS
LIN {X -0.130,Y -683.007,Z 931.423,A 0.000,B 0.000,C 90.000,E1 112.078} C_DIS
LIN {X -0.023,Y -681.311,Z 931.422,A 0.000,B 0.000,C 90.000,E1 111.950} C_DIS
LIN {X 0.062,Y -679.026,Z 931.421,A 0.000,B 0.000,C 90.000,E1 111.844} C_DIS
LIN {X -0.327,Y -674.366,Z 931.421,A 0.000,B 0.000,C 90.000,E1 111.716} C_DIS
LIN {X 0.031,Y -668.292,Z 931.420,A 0.000,B 0.000,C 90.000,E1 111.535} C_DIS
LIN {X 0.128,Y -663.611,Z 931.419,A 0.000,B 0.000,C 90.000,E1 111.482} C_DIS
LIN {X 0.126,Y -659.795,Z 931.419,A 0.000,B 0.000,C 90.000,E1 111.461} C_DIS
LIN {X 0.064,Y -640.228,Z 931.419,A 0.000,B 0.000,C 90.000,E1 111.461} C_DIS
LIN {X 0.098,Y -634.042,Z 931.419,A 0.000,B 0.000,C 90.000,E1 111.408} C_DIS
LIN {X -0.028,Y -625.642,Z 931.418,A 0.000,B 0.000,C 90.000,E1 111.280} C_DIS
LIN {X -0.061,Y -620.072,Z 931.418,A 0.000,B 0.000,C 90.000,E1 111.153} C_DIS
LIN {X 0.013,Y -614.185,Z 931.417,A 0.000,B 0.000,C 90.000,E1 110.972} C_DIS
LIN {X -0.187,Y -606.072,Z 931.415,A 0.000,B 0.000,C 90.000,E1 110.663} C_DIS
LIN {X 0.303,Y -603.125,Z 931.414,A 0.000,B 0.000,C 90.000,E1 110.482} C_DIS
LIN {X -0.292,Y -597.850,Z 931.412,A 0.000,B 0.000,C 90.000,E1 110.248} C_DIS
LIN {X -0.051,Y -589.471,Z 931.409,A 0.000,B 0.000,C 90.000,E1 109.685} C_DIS
LIN {X 0.005,Y -583.704,Z 931.407,A 0.000,B 0.000,C 90.000,E1 109.268} C_DIS
LIN {X 0.139,Y -577.745,Z 931.405,A 0.000,B 0.000,C 90.000,E1 108.852} C_DIS
LIN {X -0.009,Y -570.849,Z 931.403,A 0.000,B 0.000,C 90.000,E1 108.489} C_DIS
LIN {X 0.136,Y -565.790,Z 931.401,A 0.000,B 0.000,C 90.000,E1 108.236} C_DIS
LIN {X 0.128,Y -557.160,Z 931.399,A 0.000,B 0.000,C 90.000,E1 107.873} C_DIS
LIN {X 0.059,Y -554.737,Z 931.399,A 0.000,B 0.000,C 90.000,E1 107.764} C_DIS
LIN {X -0.262,Y -552.847,Z 931.398,A 0.000,B 0.000,C 90.000,E1 107.638} C_DIS
LIN {X 0.113,Y -552.676,Z 931.398,A 0.000,B 0.000,C 90.000,E1 107.583} C_DIS
LIN {X 0.074,Y -552.657,Z 931.398,A 0.000,B 0.000,C 90.000,E1 107.583} C_DIS
LIN {X 0.112,Y -552.206,Z 931.396,A 0.000,B 0.000,C 90.000,E1 107.347} C_DIS
LIN {X -0.039,Y -552.874,Z 931.386,A 0.000,B 0.000,C 90.000,E1 105.552} C_DIS
LIN {X -0.002,Y -553.748,Z 931.376,A 0.000,B 0.000,C 90.000,E1 103.592} C_DIS
LIN {X -0.203,Y -554.951,Z 931.365,A 0.000,B 0.000,C 90.000,E1 101.658} C_DIS
LIN {X 0.301,Y -556.726,Z 931.352,A 0.000,B 0.000,C 90.000,E1 99.378} C_DIS
LIN {X -0.166,Y -558.044,Z 931.343,A 0.000,B 0.000,C 90.000,E1 97.757} C_DIS
LIN {X 0.233,Y -558.837,Z 931.337,A 0.000,B 0.000,C 90.000,E1 96.606} C_DIS
LIN {X 0.224,Y -559.726,Z 931.329,A 0.000,B 0.000,C 90.000,E1 95.220} C_DIS
LIN {X 0.172,Y -560.508,Z 931.321,A 0.000,B 0.000,C 90.000,E1 93.841} C_DIS
LIN {X 0.099,Y -561.245,Z 931.314,A 0.000,B 0.000,C 90.000,E1 92.465} C_DIS
LIN {X 0.137,Y -561.951,Z 931.305,A 0.000,B 0.000,C 90.000,E1 90.802} C_DIS
LIN {X -0.024,Y -562.305,Z 931.298,A 0.000,B 0.000,C 90.000,E1 89.714} C_DIS
LIN {X -0.081,Y -562.662,Z 931.291,A 0.000,B 0.000,C 90.000,E1 88.339} C_DIS
LIN {X 0.010,Y -563.022,Z 931.282,A 0.000,B 0.000,C 90.000,E1 86.674} C_DIS
LIN {X 0.117,Y -563.291,Z 931.272,A 0.000,B 0.000,C 90.000,E1 85.008} C_DIS
LIN {X 0.278,Y -563.509,Z 931.263,A 0.000,B 0.000,C 90.000,E1 83.337} C_DIS
LIN {X 0.198,Y -563.723,Z 931.257,A 0.000,B 0.000,C 90.000,E1 82.243} C_DIS
LIN {X -0.130,Y -564.199,Z 931.248,A 0.000,B 0.000,C 90.000,E1 80.622} C_DIS
LIN {X -0.028,Y -565.084,Z 931.236,A 0.000,B 0.000,C 90.000,E1 78.409} C_DIS
LIN {X -0.001,Y -565.980,Z 931.227,A 0.000,B 0.000,C 90.000,E1 76.756} C_DIS
LIN {X -0.253,Y -566.891,Z 931.219,A 0.000,B 0.000,C 90.000,E1 75.408} C_DIS
LIN {X -0.204,Y -567.666,Z 931.211,A 0.000,B 0.000,C 90.000,E1 74.031} C_DIS
LIN {X 0.033,Y -568.545,Z 931.202,A 0.000,B 0.000,C 90.000,E1 72.362} C_DIS
LIN {X -0.049,Y -569.025,Z 931.196,A 0.000,B 0.000,C 90.000,E1 71.275} C_DIS
LIN {X 0.219,Y -569.645,Z 931.188,A 0.000,B 0.000,C 90.000,E1 69.880} C_DIS
LIN {X -0.226,Y -570.171,Z 931.179,A 0.000,B 0.000,C 90.000,E1 68.284} C_DIS
LIN {X 0.080,Y -570.491,Z 931.170,A 0.000,B 0.000,C 90.000,E1 66.613} C_DIS
LIN {X 0.265,Y -570.719,Z 931.163,A 0.000,B 0.000,C 90.000,E1 65.229} C_DIS
LIN {X 0.112,Y -570.997,Z 931.152,A 0.000,B 0.000,C 90.000,E1 63.332} C_DIS
LIN {X 0.039,Y -571.066,Z 931.144,A 0.000,B 0.000,C 90.000,E1 61.975} C_DIS
LIN {X -0.100,Y -571.025,Z 931.134,A 0.000,B 0.000,C 90.000,E1 60.078} C_DIS
LIN {X -0.214,Y -571.015,Z 931.128,A 0.000,B 0.000,C 90.000,E1 58.997} C_DIS
LIN {X 0.341,Y -570.920,Z 931.123,A 0.000,B 0.000,C 90.000,E1 58.122} C_DIS
LIN {X 0.299,Y -570.318,Z 931.113,A 0.000,B 0.000,C 90.000,E1 56.215} C_DIS
LIN {X -0.300,Y -569.737,Z 931.106,A 0.000,B 0.000,C 90.000,E1 55.182} C_DIS
LIN {X 0.007,Y -568.906,Z 931.099,A 0.000,B 0.000,C 90.000,E1 53.783} C_DIS
LIN {X -0.071,Y -568.228,Z 931.094,A 0.000,B 0.000,C 90.000,E1 52.970} C_DIS
LIN {X -0.372,Y -567.092,Z 931.088,A 0.000,B 0.000,C 90.000,E1 51.904} C_DIS
LIN {X -0.019,Y -566.108,Z 931.084,A 0.000,B 0.000,C 90.000,E1 51.045} C_DIS
LIN {X 0.349,Y -564.558,Z 931.078,A 0.000,B 0.000,C 90.000,E1 49.908} C_DIS
LIN {X 0.130,Y -563.750,Z 931.074,A 0.000,B 0.000,C 90.000,E1 49.380} C_DIS
LIN {X 0.002,Y -562.263,Z 931.070,A 0.000,B 0.000,C 90.000,E1 48.566} C_DIS
LIN {X -0.103,Y -559.951,Z 931.064,A 0.000,B 0.000,C 90.000,E1 47.472} C_DIS
LIN {X 0.026,Y -558.672,Z 931.061,A 0.000,B 0.000,C 90.000,E1 46.905} C_DIS
LIN {X -0.125,Y -555.720,Z 931.055,A 0.000,B 0.000,C 90.000,E1 45.810} C_DIS
LIN {X -0.024,Y -554.022,Z 931.051,A 0.000,B 0.000,C 90.000,E1 45.243} C_DIS
LIN {X -0.284,Y -551.278,Z 931.047,A 0.000,B 0.000,C 90.000,E1 44.433} C_DIS
LIN {X 0.203,Y -548.196,Z 931.042,A 0.000,B 0.000,C 90.000,E1 43.542} C_DIS
LIN {X 0.274,Y -544.709,Z 931.037,A 0.000,B 0.000,C 90.000,E1 42.690} C_DIS
LIN {X 0.117,Y -541.522,Z 931.033,A 0.000,B 0.000,C 90.000,E1 42.000} C_DIS
LIN {X 0.103,Y -538.769,Z 931.030,A 0.000,B 0.000,C 90.000,E1 41.434} C_DIS
LIN {X 0.118,Y -535.813,Z 931.027,A 0.000,B 0.000,C 90.000,E1 40.862} C_DIS
LIN {X 0.056,Y -532.628,Z 931.024,A 0.000,B 0.000,C 90.000,E1 40.297} C_DIS
LIN {X 0.014,Y -527.426,Z 931.019,A 0.000,B 0.000,C 90.000,E1 39.439} C_DIS
LIN {X 0.252,Y -522.031,Z 931.014,A 0.000,B 0.000,C 90.000,E1 38.543} C_DIS
LIN {X 0.160,Y -518.229,Z 931.011,A 0.000,B 0.000,C 90.000,E1 37.971} C_DIS
LIN {X 0.094,Y -511.108,Z 931.005,A 0.000,B 0.000,C 90.000,E1 36.950} C_DIS
LIN {X 0.029,Y -505.544,Z 931.001,A 0.000,B 0.000,C 90.000,E1 36.217} C_DIS
LIN {X -0.270,Y -502.046,Z 930.999,A 0.000,B 0.000,C 90.000,E1 35.804} C_DIS
LIN {X -0.093,Y -497.062,Z 930.995,A 0.000,B 0.000,C 90.000,E1 35.185} C_DIS
LIN {X -0.238,Y -491.855,Z 930.992,A 0.000,B 0.000,C 90.000,E1 34.612} C_DIS
LIN {X 0.215,Y -487.784,Z 930.990,A 0.000,B 0.000,C 90.000,E1 34.119} C_DIS
LIN {X -0.086,Y -482.096,Z 930.987,A 0.000,B 0.000,C 90.000,E1 33.579} C_DIS
LIN {X -0.143,Y -473.482,Z 930.982,A 0.000,B 0.000,C 90.000,E1 32.752} C_DIS
LIN {X 0.077,Y -463.235,Z 930.977,A 0.000,B 0.000,C 90.000,E1 31.799} C_DIS
LIN {X 0.114,Y -455.581,Z 930.973,A 0.000,B 0.000,C 90.000,E1 31.131} C_DIS
LIN {X -0.174,Y -444.840,Z 930.968,A 0.000,B 0.000,C 90.000,E1 30.256} C_DIS
LIN {X -0.163,Y -424.900,Z 930.959,A 0.000,B 0.000,C 90.000,E1 28.565} C_DIS
LIN {X -0.152,Y -412.708,Z 930.953,A 0.000,B 0.000,C 90.000,E1 27.462} C_DIS
LIN {X -0.131,Y -399.588,Z 930.945,A 0.000,B 0.000,C 90.000,E1 26.155} C_DIS
LIN {X 0.053,Y -395.986,Z 930.943,A 0.000,B 0.000,C 90.000,E1 25.720} C_DIS
LIN {X 0.117,Y -392.331,Z 930.940,A 0.000,B 0.000,C 90.000,E1 25.155} C_DIS
LIN {X 0.021,Y -390.300,Z 930.937,A 0.000,B 0.000,C 90.000,E1 24.695} C_DIS
LIN {X -0.037,Y -389.375,Z 930.935,A 0.000,B 0.000,C 90.000,E1 24.259} C_DIS
LIN {X -0.023,Y -389.139,Z 930.934,A 0.000,B 0.000,C 90.000,E1 24.079} C_DIS
LIN {X 0.192,Y -388.888,Z 930.931,A 0.000,B 0.000,C 90.000,E1 23.515} C_DIS
LIN {X 0.181,Y -389.150,Z 930.925,A 0.000,B 0.000,C 90.000,E1 22.461} C_DIS
LIN {X 0.186,Y -392.824,Z 930.903,A 0.000,B 0.000,C 90.000,E1 18.544} C_DIS
LIN {X 0.086,Y -395.698,Z 930.889,A 0.000,B 0.000,C 90.000,E1 16.079} C_DIS
LIN {X -0.156,Y -398.886,Z 930.876,A 0.000,B 0.000,C 90.000,E1 13.647} C_DIS
LIN {X -0.111,Y -403.035,Z 930.860,A 0.000,B 0.000,C 90.000,E1 10.838} C_DIS
LIN {X -0.094,Y -406.406,Z 930.849,A 0.000,B 0.000,C 90.000,E1 8.746} C_DIS
LIN {X -0.031,Y -410.727,Z 930.835,A 0.000,B 0.000,C 90.000,E1 6.315} C_DIS
LIN {X 0.056,Y -415.374,Z 930.822,A 0.000,B 0.000,C 90.000,E1 3.898} C_DIS
LIN {X -0.171,Y -421.261,Z 930.807,A 0.000,B 0.000,C 90.000,E1 1.203} C_DIS
LIN {X 0.211,Y -425.361,Z 930.797,A 0.000,B 0.000,C 90.000,E1 359.427} C_DIS
LIN {X 0.025,Y -428.992,Z 930.790,A 0.000,B 0.000,C 90.000,E1 358.108} C_DIS
LIN {X 0.127,Y -430.911,Z 930.787,A 0.000,B 0.000,C 90.000,E1 357.593} C_DIS
LIN {X 0.172,Y -434.330,Z 930.784,A 0.000,B 0.000,C 90.000,E1 357.020} C_DIS
LIN {X -0.222,Y -435.616,Z 930.783,A 0.000,B 0.000,C 90.000,E1 356.906} C_DIS
LIN {X -0.124,Y -437.224,Z 930.782,A 0.000,B 0.000,C 90.000,E1 356.731} C_DIS
LIN {X -0.209,Y -440.913,Z 930.780,A 0.000,B 0.000,C 90.000,E1 356.445} C_DIS
LIN {X 0.136,Y -446.668,Z 930.779,A 0.000,B 0.000,C 90.000,E1 356.102} C_DIS
LIN {X -0.051,Y -460.582,Z 930.775,A 0.000,B 0.000,C 90.000,E1 355.469} C_DIS
LIN {X -0.188,Y -468.853,Z 930.773,A 0.000,B 0.000,C 90.000,E1 355.065} C_DIS
LIN {X 0.164,Y -480.453,Z 930.769,A 0.000,B 0.000,C 90.000,E1 354.432} C_DIS
LIN {X 0.129,Y -487.195,Z 930.767,A 0.000,B 0.000,C 90.000,E1 354.090} C_DIS
LIN {X 0.052,Y -500.020,Z 930.763,A 0.000,B 0.000,C 90.000,E1 353.394} C_DIS
LIN {X 0.123,Y -509.733,Z 930.760,A 0.000,B 0.000,C 90.000,E1 352.818} C_DIS
LIN {X -0.086,Y -519.235,Z 930.757,A 0.000,B 0.000,C 90.000,E1 352.243} C_DIS
LIN {X -0.167,Y -525.549,Z 930.755,A 0.000,B 0.000,C 90.000,E1 351.837} C_DIS
LIN {X 0.245,Y -532.829,Z 930.752,A 0.000,B 0.000,C 90.000,E1 351.254} C_DIS
LIN {X -0.272,Y -537.112,Z 930.750,A 0.000,B 0.000,C 90.000,E1 350.971} C_DIS
LIN {X 0.228,Y -542.821,Z 930.747,A 0.000,B 0.000,C 90.000,E1 350.443} C_DIS
LIN {X -0.196,Y -549.688,Z 930.744,A 0.000,B 0.000,C 90.000,E1 349.859} C_DIS
LIN {X -0.219,Y -554.915,Z 930.741,A 0.000,B 0.000,C 90.000,E1 349.342} C_DIS
LIN {X -0.265,Y -559.825,Z 930.738,A 0.000,B 0.000,C 90.000,E1 348.814} C_DIS
LIN {X 0.055,Y -567.742,Z 930.732,A 0.000,B 0.000,C 90.000,E1 347.825} C_DIS
LIN {X -0.269,Y -572.961,Z 930.729,A 0.000,B 0.000,C 90.000,E1 347.173} C_DIS
LIN {X 0.225,Y -579.714,Z 930.723,A 0.000,B 0.000,C 90.000,E1 346.172} C_DIS
LIN {X 0.104,Y -583.211,Z 930.720,A 0.000,B 0.000,C 90.000,E1 345.644} C_DIS
LIN {X 0.160,Y -589.024,Z 930.715,A 0.000,B 0.000,C 90.000,E1 344.700} C_DIS
LIN {X -0.125,Y -594.364,Z 930.710,A 0.000,B 0.000,C 90.000,E1 343.795} C_DIS
LIN {X -0.001,Y -599.882,Z 930.704,A 0.000,B 0.000,C 90.000,E1 342.725} C_DIS
LIN {X 0.145,Y -605.687,Z 930.698,A 0.000,B 0.000,C 90.000,E1 341.529} C_DIS
LIN {X 0.294,Y -609.467,Z 930.693,A 0.000,B 0.000,C 90.000,E1 340.732} C_DIS
LIN {X -0.321,Y -613.684,Z 930.688,A 0.000,B 0.000,C 90.000,E1 339.880} C_DIS
LIN {X -0.121,Y -618.121,Z 930.682,A 0.000,B 0.000,C 90.000,E1 338.827} C_DIS
LIN {X -0.083,Y -622.298,Z 930.677,A 0.000,B 0.000,C 90.000,E1 337.794} C_DIS
LIN {X 0.240,Y -626.247,Z 930.671,A 0.000,B 0.000,C 90.000,E1 336.741} C_DIS
LIN {X 0.020,Y -628.973,Z 930.667,A 0.000,B 0.000,C 90.000,E1 335.997} C_DIS
LIN {X 0.086,Y -631.664,Z 930.662,A 0.000,B 0.000,C 90.000,E1 335.229} C_DIS
LIN {X -0.010,Y -635.765,Z 930.655,A 0.000,B 0.000,C 90.000,E1 333.973} C_DIS
LIN {X 0.181,Y -638.884,Z 930.650,A 0.000,B 0.000,C 90.000,E1 332.948} C_DIS
LIN {X 0.282,Y -643.068,Z 930.641,A 0.000,B 0.000,C 90.000,E1 331.435} C_DIS
LIN {X 0.005,Y -645.481,Z 930.636,A 0.000,B 0.000,C 90.000,E1 330.461} C_DIS
LIN {X 0.158,Y -648.515,Z 930.629,A 0.000,B 0.000,C 90.000,E1 329.203} C_DIS
LIN {X -0.199,Y -651.116,Z 930.622,A 0.000,B 0.000,C 90.000,E1 327.995} C_DIS
LIN {X -0.164,Y -653.296,Z 930.615,A 0.000,B 0.000,C 90.000,E1 326.755} C_DIS
LIN {X -0.088,Y -654.424,Z 930.611,A 0.000,B 0.000,C 90.000,E1 326.008} C_DIS
LIN {X -0.085,Y -655.750,Z 930.606,A 0.000,B 0.000,C 90.000,E1 325.022} C_DIS
LIN {X 0.006,Y -656.719,Z 930.602,A 0.000,B 0.000,C 90.000,E1 324.276} C_DIS
LIN {X 0.048,Y -658.268,Z 930.593,A 0.000,B 0.000,C 90.000,E1 322.798} C_DIS
LIN {X -0.030,Y -659.048,Z 930.588,A 0.000,B 0.000,C 90.000,E1 321.823} C_DIS
LIN {X -0.026,Y -660.050,Z 930.581,A 0.000,B 0.000,C 90.000,E1 320.598} C_DIS
LIN {X 0.352,Y -661.421,Z 930.572,A 0.000,B 0.000,C 90.000,E1 318.852} C_DIS
LIN {X 0.305,Y -662.477,Z 930.565,A 0.000,B 0.000,C 90.000,E1 317.634} C_DIS
LIN {X -0.228,Y -663.824,Z 930.557,A 0.000,B 0.000,C 90.000,E1 316.215} C_DIS
LIN {X -0.267,Y -664.707,Z 930.550,A 0.000,B 0.000,C 90.000,E1 315.000} C_DIS
LIN {X 0.186,Y -666.467,Z 930.539,A 0.000,B 0.000,C 90.000,E1 313.014} C_DIS
LIN {X 0.227,Y -668.087,Z 930.530,A 0.000,B 0.000,C 90.000,E1 311.310} C_DIS
LIN {X -0.140,Y -669.428,Z 930.522,A 0.000,B 0.000,C 90.000,E1 309.886} C_DIS
LIN {X -0.060,Y -670.510,Z 930.515,A 0.000,B 0.000,C 90.000,E1 308.669} C_DIS
LIN {X -0.284,Y -671.568,Z 930.507,A 0.000,B 0.000,C 90.000,E1 307.237} C_DIS
LIN {X -0.057,Y -672.082,Z 930.501,A 0.000,B 0.000,C 90.000,E1 306.251} C_DIS
LIN {X 0.017,Y -672.836,Z 930.489,A 0.000,B 0.000,C 90.000,E1 304.072} C_DIS
LIN {X 0.123,Y -673.760,Z 930.479,A 0.000,B 0.000,C 90.000,E1 302.133} C_DIS
LIN {X -0.122,Y -675.387,Z 930.465,A 0.000,B 0.000,C 90.000,E1 299.745} C_DIS
LIN {X -0.170,Y -680.742,Z 930.443,A 0.000,B 0.000,C 90.000,E1 295.668} C_DIS
LIN {X 0.025,Y -682.218,Z 930.437,A 0.000,B 0.000,C 90.000,E1 294.695} C_DIS
LIN {X -0.333,Y -683.529,Z 930.432,A 0.000,B 0.000,C 90.000,E1 293.770} C_DIS
LIN {X 0.023,Y -684.264,Z 930.428,A 0.000,B 0.000,C 90.000,E1 293.025} C_DIS
LIN {X -0.191,Y -684.369,Z 930.425,A 0.000,B 0.000,C 90.000,E1 292.567} C_DIS
LIN {X -0.245,Y -684.181,Z 930.424,A 0.000,B 0.000,C 90.000,E1 292.333} C_DIS
LIN {X -0.089,Y -683.308,Z 930.421,A 0.000,B 0.000,C 90.000,E1 291.844} C_DIS
LIN {X 0.114,Y -682.246,Z 930.420,A 0.000,B 0.000,C 90.000,E1 291.589} C_DIS
LIN {X 0.214,Y -681.252,Z 930.419,A 0.000,B 0.000,C 90.000,E1 291.461} C_DIS
LIN {X 0.183,Y -678.867,Z 930.418,A 0.000,B 0.000,C 90.000,E1 291.227} C_DIS
LIN {X 0.300,Y -677.902,Z 930.417,A 0.000,B 0.000,C 90.000,E1 291.099} C_DIS
LIN {X 0.391,Y -676.727,Z 930.417,A 0.000,B 0.000,C 90.000,E1 290.972} C_DIS
LIN {X -0.041,Y -673.350,Z 930.416,A 0.000,B 0.000,C 90.000,E1 290.791} C_DIS
LIN {X 0.102,Y -664.097,Z 930.413,A 0.000,B 0.000,C 90.000,E1 290.248} C_DIS
LIN {X -0.255,Y -662.160,Z 930.412,A 0.000,B 0.000,C 90.000,E1 290.120} C_DIS
LIN {X -0.322,Y -662.120,Z 930.412,A 0.000,B 0.000,C 90.000,E1 290.120} C_DIS
LIN {X 0.159,Y -661.850,Z 930.411,A 0.000,B 0.000,C 90.000,E1 289.939} C_DIS
LIN {X 0.218,Y -661.952,Z 930.410,A 0.000,B 0.000,C 90.000,E1 289.812} C_DIS
LIN {X 0.169,Y -662.783,Z 930.408,A 0.000,B 0.000,C 90.000,E1 289.450} C_DIS
LIN {X 0.125,Y -664.211,Z 930.406,A 0.000,B 0.000,C 90.000,E1 289.087} C_DIS
LIN {X 0.158,Y -669.710,Z 930.400,A 0.000,B 0.000,C 90.000,E1 288.000} C_DIS
LIN {X 0.077,Y -672.777,Z 930.397,A 0.000,B 0.000,C 90.000,E1 287.402} C_DIS
LIN {X 0.145,Y -675.037,Z 930.394,A 0.000,B 0.000,C 90.000,E1 286.913} C_DIS
LIN {X 0.030,Y -677.024,Z 930.391,A 0.000,B 0.000,C 90.000,E1 286.441} C_DIS
LIN {X 0.072,Y -679.472,Z 930.387,A 0.000,B 0.000,C 90.000,E1 285.717} C_DIS
LIN {X -0.047,Y -681.352,Z 930.383,A 0.000,B 0.000,C 90.000,E1 285.009} C_DIS
LIN {X -0.174,Y -683.485,Z 930.378,A 0.000,B 0.000,C 90.000,E1 284.064} C_DIS
LIN {X -0.276,Y -685.104,Z 930.373,A 0.000,B 0.000,C 90.000,E1 283.119} C_DIS
LIN {X 0.328,Y -686.114,Z 930.369,A 0.000,B 0.000,C 90.000,E1 282.355} C_DIS
LIN {X 0.129,Y -686.839,Z 930.365,A 0.000,B 0.000,C 90.000,E1 281.658} C_DIS
LIN {X 0.094,Y -687.133,Z 930.362,A 0.000,B 0.000,C 90.000,E1 281.186} C_DIS
LIN {X 0.056,Y -687.099,Z 930.360,A 0.000,B 0.000,C 90.000,E1 280.715} C_DIS
LIN {X -0.110,Y -686.762,Z 930.357,A 0.000,B 0.000,C 90.000,E1 280.254} C_DIS
LIN {X -0.131,Y -686.482,Z 930.356,A 0.000,B 0.000,C 90.000,E1 280.018} C_DIS
LIN {X -0.294,Y -685.573,Z 930.353,A 0.000,B 0.000,C 90.000,E1 279.557} C_DIS
LIN {X 0.324,Y -684.175,Z 930.350,A 0.000,B 0.000,C 90.000,E1 279.029} C_DIS
LIN {X 0.150,Y -682.382,Z 930.348,A 0.000,B 0.000,C 90.000,E1 278.568} C_DIS
LIN {X 0.010,Y -681.371,Z 930.346,A 0.000,B 0.000,C 90.000,E1 278.341} C_DIS
LIN {X -0.282,Y -676.664,Z 930.341,A 0.000,B 0.000,C 90.000,E1 277.409} C_DIS
LIN {X -0.067,Y -671.536,Z 930.336,A 0.000,B 0.000,C 90.000,E1 276.429} C_DIS
LIN {X 0.263,Y -667.948,Z 930.332,A 0.000,B 0.000,C 90.000,E1 275.796} C_DIS
LIN {X -0.099,Y -663.672,Z 930.329,A 0.000,B 0.000,C 90.000,E1 275.220} C_DIS
LIN {X 0.257,Y -659.902,Z 930.326,A 0.000,B 0.000,C 90.000,E1 274.702} C_DIS
LIN {X -0.120,Y -655.779,Z 930.324,A 0.000,B 0.000,C 90.000,E1 274.245} C_DIS
LIN {X 0.179,Y -650.220,Z 930.320,A 0.000,B 0.000,C 90.000,E1 273.612} C_DIS
LIN {X -0.158,Y -645.381,Z 930.318,A 0.000,B 0.000,C 90.000,E1 273.154} C_DIS
LIN {X -0.311,Y -638.828,Z 930.314,A 0.000,B 0.000,C 90.000,E1 272.579} C_DIS
LIN {X -0.153,Y -631.838,Z 930.311,A 0.000,B 0.000,C 90.000,E1 272.007} C_DIS
LIN {X -0.240,Y -624.388,Z 930.308,A 0.000,B 0.000,C 90.000,E1 271.489} C_DIS
LIN {X -0.024,Y -616.543,Z 930.305,A 0.000,B 0.000,C 90.000,E1 270.974} C_DIS
LIN {X 0.279,Y -610.204,Z 930.303,A 0.000,B 0.000,C 90.000,E1 270.573} C_DIS
LIN {X 0.250,Y -603.592,Z 930.301,A 0.000,B 0.000,C 90.000,E1 270.229} C_DIS
LIN {X -0.133,Y -596.759,Z 930.300,A 0.000,B 0.000,C 90.000,E1 269.943} C_DIS
LIN {X -0.079,Y -591.447,Z 930.298,A 0.000,B 0.000,C 90.000,E1 269.714} C_DIS
LIN {X 0.121,Y -584.058,Z 930.297,A 0.000,B 0.000,C 90.000,E1 269.427} C_DIS
LIN {X 0.117,Y -578.191,Z 930.296,A 0.000,B 0.000,C 90.000,E1 269.255} C_DIS
LIN {X 0.011,Y -570.372,Z 930.295,A 0.000,B 0.000,C 90.000,E1 269.083} C_DIS
LIN {X 0.085,Y -564.553,Z 930.294,A 0.000,B 0.000,C 90.000,E1 268.969} C_DIS
LIN {X -0.028,Y -557.785,Z 930.294,A 0.000,B 0.000,C 90.000,E1 268.912} C_DIS
LIN {X 0.119,Y -552.066,Z 930.294,A 0.000,B 0.000,C 90.000,E1 268.854} C_DIS
LIN {X -0.100,Y -550.980,Z 930.294,A 0.000,B 0.000,C 90.000,E1 268.854} C_DIS
LIN {X -0.145,Y -550.844,Z 930.294,A 0.000,B 0.000,C 90.000,E1 268.854} C_DIS
LIN {X 0.028,Y -549.391,Z 930.292,A 0.000,B 0.000,C 90.000,E1 268.625} C_DIS
LIN {X -0.165,Y -545.767,Z 930.290,A 0.000,B 0.000,C 90.000,E1 268.224} C_DIS
LIN {X 0.104,Y -544.180,Z 930.289,A 0.000,B 0.000,C 90.000,E1 268.051} C_DIS
LIN {X 0.062,Y -544.157,Z 930.289,A 0.000,B 0.000,C 90.000,E1 268.051} C_DIS
LIN {X 0.184,Y -543.442,Z 930.288,A 0.000,B 0.000,C 90.000,E1 267.764} C_DIS
LIN {X -0.149,Y -540.042,Z 930.266,A 0.000,B 0.000,C 90.000,E1 263.970} C_DIS
LIN {X 0.044,Y -538.913,Z 930.257,A 0.000,B 0.000,C 90.000,E1 262.243} C_DIS
LIN {X -0.243,Y -537.879,Z 930.249,A 0.000,B 0.000,C 90.000,E1 260.849} C_DIS
LIN {X -0.141,Y -537.062,Z 930.244,A 0.000,B 0.000,C 90.000,E1 259.982} C_DIS
LIN {X 0.102,Y -535.535,Z 930.238,A 0.000,B 0.000,C 90.000,E1 258.814} C_DIS
LIN {X -0.008,Y -532.452,Z 930.225,A 0.000,B 0.000,C 90.000,E1 256.533} C_DIS
LIN {X -0.028,Y -530.357,Z 930.216,A 0.000,B 0.000,C 90.000,E1 254.810} C_DIS
LIN {X -0.109,Y -528.626,Z 930.208,A 0.000,B 0.000,C 90.000,E1 253.378} C_DIS
LIN {X -0.225,Y -526.835,Z 930.200,A 0.000,B 0.000,C 90.000,E1 251.945} C_DIS
LIN {X -0.053,Y -524.586,Z 930.190,A 0.000,B 0.000,C 90.000,E1 250.188} C_DIS
LIN {X -0.072,Y -523.127,Z 930.183,A 0.000,B 0.000,C 90.000,E1 249.028} C_DIS
LIN {X 0.234,Y -521.231,Z 930.175,A 0.000,B 0.000,C 90.000,E1 247.539} C_DIS
LIN {X 0.029,Y -519.143,Z 930.167,A 0.000,B 0.000,C 90.000,E1 246.102} C_DIS
LIN {X 0.265,Y -515.941,Z 930.156,A 0.000,B 0.000,C 90.000,E1 244.024} C_DIS
LIN {X 0.058,Y -514.093,Z 930.149,A 0.000,B 0.000,C 90.000,E1 242.871} C_DIS
LIN {X -0.190,Y -511.108,Z 930.140,A 0.000,B 0.000,C 90.000,E1 241.129} C_DIS
LIN {X 0.024,Y -509.056,Z 930.133,A 0.000,B 0.000,C 90.000,E1 239.921} C_DIS
LIN {X -0.047,Y -506.908,Z 930.126,A 0.000,B 0.000,C 90.000,E1 238.742} C_DIS
LIN {X -0.211,Y -505.151,Z 930.121,A 0.000,B 0.000,C 90.000,E1 237.867} C_DIS
LIN {X 0.186,Y -502.584,Z 930.115,A 0.000,B 0.000,C 90.000,E1 236.628} C_DIS
LIN {X -0.152,Y -499.821,Z 930.108,A 0.000,B 0.000,C 90.000,E1 235.468} C_DIS
LIN {X 0.046,Y -495.092,Z 930.096,A 0.000,B 0.000,C 90.000,E1 233.336} C_DIS
LIN {X 0.029,Y -491.865,Z 930.088,A 0.000,B 0.000,C 90.000,E1 231.823} C_DIS
LIN {X 0.103,Y -489.145,Z 930.081,A 0.000,B 0.000,C 90.000,E1 230.598} C_DIS
LIN {X 0.036,Y -484.991,Z 930.071,A 0.000,B 0.000,C 90.000,E1 228.771} C_DIS
LIN {X 0.075,Y -481.480,Z 930.063,A 0.000,B 0.000,C 90.000,E1 227.229} C_DIS
LIN {X 0.038,Y -478.048,Z 930.054,A 0.000,B 0.000,C 90.000,E1 225.688} C_DIS
LIN {X 0.260,Y -474.690,Z 930.045,A 0.000,B 0.000,C 90.000,E1 224.109} C_DIS
LIN {X -0.244,Y -471.219,Z 930.037,A 0.000,B 0.000,C 90.000,E1 222.609} C_DIS
LIN {X 0.196,Y -467.751,Z 930.028,A 0.000,B 0.000,C 90.000,E1 220.987} C_DIS
LIN {X 0.167,Y -462.294,Z 930.014,A 0.000,B 0.000,C 90.000,E1 218.463} C_DIS
LIN {X 0.192,Y -458.898,Z 930.005,A 0.000,B 0.000,C 90.000,E1 216.870} C_DIS
LIN {X -0.121,Y -455.440,Z 929.996,A 0.000,B 0.000,C 90.000,E1 215.311} C_DIS
LIN {X -0.129,Y -451.888,Z 929.987,A 0.000,B 0.000,C 90.000,E1 213.706} C_DIS
LIN {X 0.078,Y -446.927,Z 929.975,A 0.000,B 0.000,C 90.000,E1 211.416} C_DIS
LIN {X -0.025,Y -441.202,Z 929.960,A 0.000,B 0.000,C 90.000,E1 208.821} C_DIS
LIN {X -0.031,Y -437.668,Z 929.951,A 0.000,B 0.000,C 90.000,E1 207.180} C_DIS
LIN {X -0.114,Y -434.012,Z 929.942,A 0.000,B 0.000,C 90.000,E1 205.540} C_DIS
LIN {X -0.066,Y -428.917,Z 929.929,A 0.000,B 0.000,C 90.000,E1 203.206} C_DIS
LIN {X 0.111,Y -425.990,Z 929.922,A 0.000,B 0.000,C 90.000,E1 201.844} C_DIS
LIN {X 0.024,Y -422.287,Z 929.912,A 0.000,B 0.000,C 90.000,E1 200.174} C_DIS
LIN {X 0.226,Y -416.163,Z 929.895,A 0.000,B 0.000,C 90.000,E1 197.094} C_DIS
LIN {X 0.162,Y -414.122,Z 929.890,A 0.000,B 0.000,C 90.000,E1 196.079} C_DIS
LIN {X 0.228,Y -410.572,Z 929.880,A 0.000,B 0.000,C 90.000,E1 194.356} C_DIS
LIN {X 0.013,Y -407.793,Z 929.872,A 0.000,B 0.000,C 90.000,E1 193.008} C_DIS
LIN {X -0.141,Y -402.996,Z 929.859,A 0.000,B 0.000,C 90.000,E1 190.602} C_DIS
LIN {X -0.187,Y -398.270,Z 929.845,A 0.000,B 0.000,C 90.000,E1 188.163} C_DIS
LIN {X -0.084,Y -393.428,Z 929.832,A 0.000,B 0.000,C 90.000,E1 185.682} C_DIS
LIN {X 0.132,Y -388.239,Z 929.816,A 0.000,B 0.000,C 90.000,E1 182.808} C_DIS
LIN {X -0.096,Y -382.570,Z 929.796,A 0.000,B 0.000,C 90.000,E1 179.255} C_DIS
LIN {X -0.165,Y -381.006,Z 929.788,A 0.000,B 0.000,C 90.000,E1 177.822} C_DIS
LIN {X -0.027,Y -380.674,Z 929.784,A 0.000,B 0.000,C 90.000,E1 177.078} C_DIS
LIN {X -0.130,Y -380.509,Z 929.782,A 0.000,B 0.000,C 90.000,E1 176.731} C_DIS
LIN {X -0.003,Y -380.656,Z 929.778,A 0.000,B 0.000,C 90.000,E1 175.988} C_DIS
LIN {X -0.103,Y -381.044,Z 929.776,A 0.000,B 0.000,C 90.000,E1 175.641} C_DIS
LIN {X 0.148,Y -381.681,Z 929.774,A 0.000,B 0.000,C 90.000,E1 175.241} C_DIS
LIN {X 0.126,Y -382.495,Z 929.772,A 0.000,B 0.000,C 90.000,E1 174.894} C_DIS
LIN {X -0.027,Y -384.567,Z 929.769,A 0.000,B 0.000,C 90.000,E1 174.375} C_DIS
LIN {X -0.089,Y -385.452,Z 929.768,A 0.000,B 0.000,C 90.000,E1 174.204} C_DIS
LIN {X -0.077,Y -389.051,Z 929.765,A 0.000,B 0.000,C 90.000,E1 173.628} C_DIS
LIN {X -0.096,Y -395.530,Z 929.761,A 0.000,B 0.000,C 90.000,E1 172.932} C_DIS
LIN {X -0.016,Y -401.499,Z 929.758,A 0.000,B 0.000,C 90.000,E1 172.413} C_DIS
LIN {X -0.106,Y -412.624,Z 929.753,A 0.000,B 0.000,C 90.000,E1 171.602} C_DIS
LIN {X 0.191,Y -417.395,Z 929.751,A 0.000,B 0.000,C 90.000,E1 171.197} C_DIS
LIN {X -0.082,Y -426.360,Z 929.747,A 0.000,B 0.000,C 90.000,E1 170.557} C_DIS
LIN {X -0.125,Y -437.339,Z 929.743,A 0.000,B 0.000,C 90.000,E1 169.690} C_DIS
LIN {X 0.151,Y -446.280,Z 929.738,A 0.000,B 0.000,C 90.000,E1 168.870} C_DIS
LIN {X -0.125,Y -453.773,Z 929.735,A 0.000,B 0.000,C 90.000,E1 168.229} C_DIS
LIN {X -0.039,Y -460.918,Z 929.731,A 0.000,B 0.000,C 90.000,E1 167.521} C_DIS
LIN {X -0.231,Y -467.928,Z 929.727,A 0.000,B 0.000,C 90.000,E1 166.825} C_DIS
LIN {X -0.042,Y -474.654,Z 929.723,A 0.000,B 0.000,C 90.000,E1 166.061} C_DIS
LIN {X 0.092,Y -478.569,Z 929.720,A 0.000,B 0.000,C 90.000,E1 165.589} C_DIS
LIN {X -0.202,Y -487.437,Z 929.714,A 0.000,B 0.000,C 90.000,E1 164.574} C_DIS
LIN {X -0.066,Y -493.479,Z 929.710,A 0.000,B 0.000,C 90.000,E1 163.795} C_DIS
LIN {X 0.058,Y -501.244,Z 929.704,A 0.000,B 0.000,C 90.000,E1 162.725} C_DIS
LIN {X -0.201,Y -513.603,Z 929.694,A 0.000,B 0.000,C 90.000,E1 160.967} C_DIS
LIN {X -0.173,Y -520.528,Z 929.688,A 0.000,B 0.000,C 90.000,E1 159.934} C_DIS
LIN {X 0.112,Y -528.967,Z 929.681,A 0.000,B 0.000,C 90.000,E1 158.592} C_DIS
LIN {X -0.313,Y -536.160,Z 929.675,A 0.000,B 0.000,C 90.000,E1 157.486} C_DIS
LIN {X 0.039,Y -546.534,Z 929.665,A 0.000,B 0.000,C 90.000,E1 155.741} C_DIS
LIN {X 0.042,Y -549.811,Z 929.662,A 0.000,B 0.000,C 90.000,E1 155.177} C_DIS
LIN {X 0.137,Y -557.732,Z 929.654,A 0.000,B 0.000,C 90.000,E1 153.768} C_DIS
LIN {X 0.012,Y -562.102,Z 929.650,A 0.000,B 0.000,C 90.000,E1 152.948} C_DIS
LIN {X 0.002,Y -567.742,Z 929.644,A 0.000,B 0.000,C 90.000,E1 151.847} C_DIS
LIN {X 0.100,Y -574.888,Z 929.635,A 0.000,B 0.000,C 90.000,E1 150.333} C_DIS
LIN {X -0.021,Y -580.236,Z 929.628,A 0.000,B 0.000,C 90.000,E1 149.125} C_DIS
LIN {X -0.013,Y -582.576,Z 929.625,A 0.000,B 0.000,C 90.000,E1 148.584} C_DIS
LIN {X 0.105,Y -589.038,Z 929.617,A 0.000,B 0.000,C 90.000,E1 146.962} C_DIS
LIN {X -0.360,Y -594.305,Z 929.609,A 0.000,B 0.000,C 90.000,E1 145.674} C_DIS
LIN {X -0.040,Y -597.413,Z 929.605,A 0.000,B 0.000,C 90.000,E1 144.848} C_DIS
LIN {X -0.177,Y -600.396,Z 929.600,A 0.000,B 0.000,C 90.000,E1 144.069} C_DIS
LIN {X 0.267,Y -607.022,Z 929.590,A 0.000,B 0.000,C 90.000,E1 142.190} C_DIS
LIN {X 0.405,Y -613.850,Z 929.580,A 0.000,B 0.000,C 90.000,E1 140.356} C_DIS
LIN {X -0.082,Y -619.827,Z 929.571,A 0.000,B 0.000,C 90.000,E1 138.852} C_DIS
LIN {X -0.108,Y -629.825,Z 929.557,A 0.000,B 0.000,C 90.000,E1 136.296} C_DIS
LIN {X 0.322,Y -633.912,Z 929.552,A 0.000,B 0.000,C 90.000,E1 135.243} C_DIS
LIN {X -0.183,Y -638.796,Z 929.545,A 0.000,B 0.000,C 90.000,E1 134.028} C_DIS
LIN {X -0.152,Y -643.691,Z 929.538,A 0.000,B 0.000,C 90.000,E1 132.771} C_DIS
LIN {X 0.315,Y -650.494,Z 929.528,A 0.000,B 0.000,C 90.000,E1 130.987} C_DIS
LIN {X -0.232,Y -652.474,Z 929.525,A 0.000,B 0.000,C 90.000,E1 130.539} C_DIS
LIN {X -0.420,Y -658.994,Z 929.516,A 0.000,B 0.000,C 90.000,E1 128.830} C_DIS
LIN {X 0.079,Y -661.824,Z 929.511,A 0.000,B 0.000,C 90.000,E1 128.051} C_DIS
LIN {X 0.124,Y -667.353,Z 929.503,A 0.000,B 0.000,C 90.000,E1 126.583} C_DIS
LIN {X 0.302,Y -670.896,Z 929.498,A 0.000,B 0.000,C 90.000,E1 125.598} C_DIS
LIN {X -0.003,Y -673.453,Z 929.494,A 0.000,B 0.000,C 90.000,E1 124.898} C_DIS
LIN {X 0.253,Y -676.654,Z 929.489,A 0.000,B 0.000,C 90.000,E1 123.913} C_DIS
LIN {X 0.170,Y -679.572,Z 929.483,A 0.000,B 0.000,C 90.000,E1 122.959} C_DIS
LIN {X -0.064,Y -681.522,Z 929.479,A 0.000,B 0.000,C 90.000,E1 122.260} C_DIS
LIN {X -0.064,Y -683.335,Z 929.475,A 0.000,B 0.000,C 90.000,E1 121.544} C_DIS
LIN {X 0.144,Y -685.949,Z 929.469,A 0.000,B 0.000,C 90.000,E1 120.335} C_DIS
LIN {X -0.019,Y -686.874,Z 929.466,A 0.000,B 0.000,C 90.000,E1 119.873} C_DIS
LIN {X -0.101,Y -688.885,Z 929.459,A 0.000,B 0.000,C 90.000,E1 118.693} C_DIS
LIN {X -0.247,Y -689.567,Z 929.457,A 0.000,B 0.000,C 90.000,E1 118.231} C_DIS
LIN {X -0.156,Y -690.370,Z 929.453,A 0.000,B 0.000,C 90.000,E1 117.513} C_DIS
LIN {X 0.176,Y -691.024,Z 929.448,A 0.000,B 0.000,C 90.000,E1 116.539} C_DIS
LIN {X -0.033,Y -691.244,Z 929.444,A 0.000,B 0.000,C 90.000,E1 115.848} C_DIS
LIN {X 0.005,Y -691.335,Z 929.438,A 0.000,B 0.000,C 90.000,E1 114.899} C_DIS
LIN {X -0.433,Y -691.273,Z 929.436,A 0.000,B 0.000,C 90.000,E1 114.463} C_DIS
LIN {X 0.043,Y -691.014,Z 929.433,A 0.000,B 0.000,C 90.000,E1 113.951} C_DIS
LIN {X 0.238,Y -690.549,Z 929.430,A 0.000,B 0.000,C 90.000,E1 113.462} C_DIS
LIN {X -0.162,Y -690.019,Z 929.429,A 0.000,B 0.000,C 90.000,E1 113.259} C_DIS
LIN {X 0.029,Y -688.476,Z 929.427,A 0.000,B 0.000,C 90.000,E1 112.770} C_DIS
LIN {X 0.141,Y -687.811,Z 929.426,A 0.000,B 0.000,C 90.000,E1 112.642} C_DIS
LIN {X 0.101,Y -686.087,Z 929.425,A 0.000,B 0.000,C 90.000,E1 112.408} C_DIS
LIN {X -0.315,Y -683.900,Z 929.423,A 0.000,B 0.000,C 90.000,E1 112.206} C_DIS
LIN {X -0.209,Y -682.687,Z 929.423,A 0.000,B 0.000,C 90.000,E1 112.078} C_DIS
LIN {X -0.088,Y -680.924,Z 929.422,A 0.000,B 0.000,C 90.000,E1 111.950} C_DIS
LIN {X -0.220,Y -678.102,Z 929.421,A 0.000,B 0.000,C 90.000,E1 111.844} C_DIS
LIN {X -0.137,Y -672.225,Z 929.420,A 0.000,B 0.000,C 90.000,E1 111.642} C_DIS
LIN {X -0.047,Y -668.415,Z 929.420,A 0.000,B 0.000,C 90.000,E1 111.535} C_DIS
LIN {X -0.030,Y -660.489,Z 929.419,A 0.000,B 0.000,C 90.000,E1 111.461} C_DIS
LIN {X -0.080,Y -643.179,Z 929.419,A 0.000,B 0.000,C 90.000,E1 111.461} C_DIS
LIN {X 0.159,Y -637.398,Z 929.419,A 0.000,B 0.000,C 90.000,E1 111.408} C_DIS
LIN {X -0.153,Y -633.983,Z 929.419,A 0.000,B 0.000,C 90.000,E1 111.408} C_DIS
LIN {X 0.311,Y -628.565,Z 929.418,A 0.000,B 0.000,C 90.000,E1 111.280} C_DIS
LIN {X -0.018,Y -621.232,Z 929.418,A 0.000,B 0.000,C 90.000,E1 111.153} C_DIS
LIN {X 0.216,Y -613.930,Z 929.416,A 0.000,B 0.000,C 90.000,E1 110.918} C_DIS
LIN {X -0.033,Y -605.813,Z 929.415,A 0.000,B 0.000,C 90.000,E1 110.610} C_DIS
LIN {X -0.115,Y -602.915,Z 929.414,A 0.000,B 0.000,C 90.000,E1 110.482} C_DIS
LIN {X -0.211,Y -596.339,Z 929.412,A 0.000,B 0.000,C 90.000,E1 110.120} C_DIS
LIN {X -0.087,Y -589.052,Z 929.409,A 0.000,B 0.000,C 90.000,E1 109.631} C_DIS
LIN {X 0.119,Y -581.551,Z 929.406,A 0.000,B 0.000,C 90.000,E1 109.087} C_DIS
LIN {X -0.127,Y -578.551,Z 929.405,A 0.000,B 0.000,C 90.000,E1 108.906} C_DIS
LIN {X -0.228,Y -571.745,Z 929.403,A 0.000,B 0.000,C 90.000,E1 108.544} C_DIS
LIN {X 0.262,Y -566.337,Z 929.401,A 0.000,B 0.000,C 90.000,E1 108.236} C_DIS
LIN {X 0.102,Y -556.178,Z 929.399,A 0.000,B 0.000,C 90.000,E1 107.819} C_DIS
LIN {X -0.141,Y -554.559,Z 929.399,A 0.000,B 0.000,C 90.000,E1 107.764} C_DIS
LIN {X 0.081,Y -552.836,Z 929.398,A 0.000,B 0.000,C 90.000,E1 107.583} C_DIS
LIN {X 0.044,Y -552.809,Z 929.398,A 0.000,B 0.000,C 90.000,E1 107.583} C_DIS
LIN {X 0.164,Y -552.479,Z 929.397,A 0.000,B 0.000,C 90.000,E1 107.402} C_DIS
LIN {X 0.011,Y -552.419,Z 929.394,A 0.000,B 0.000,C 90.000,E1 106.858} C_DIS
LIN {X 0.078,Y -552.939,Z 929.388,A 0.000,B 0.000,C 90.000,E1 105.733} C_DIS
LIN {X -0.001,Y -553.669,Z 929.378,A 0.000,B 0.000,C 90.000,E1 104.064} C_DIS
LIN {X 0.040,Y -554.953,Z 929.366,A 0.000,B 0.000,C 90.000,E1 101.827} C_DIS
LIN {X 0.025,Y -556.904,Z 929.352,A 0.000,B 0.000,C 90.000,E1 99.321} C_DIS
LIN {X 0.117,Y -558.204,Z 929.343,A 0.000,B 0.000,C 90.000,E1 97.644} C_DIS
LIN {X -0.034,Y -558.988,Z 929.336,A 0.000,B 0.000,C 90.000,E1 96.549} C_DIS
LIN {X 0.042,Y -560.031,Z 929.327,A 0.000,B 0.000,C 90.000,E1 94.878} C_DIS
LIN {X 0.001,Y -560.764,Z 929.319,A 0.000,B 0.000,C 90.000,E1 93.498} C_DIS
LIN {X -0.159,Y -561.352,Z 929.313,A 0.000,B 0.000,C 90.000,E1 92.407} C_DIS
LIN {X -0.118,Y -562.053,Z 929.304,A 0.000,B 0.000,C 90.000,E1 90.745} C_DIS
LIN {X -0.278,Y -562.384,Z 929.298,A 0.000,B 0.000,C 90.000,E1 89.656} C_DIS
LIN {X 0.228,Y -562.741,Z 929.290,A 0.000,B 0.000,C 90.000,E1 88.224} C_DIS
LIN {X -0.144,Y -563.132,Z 929.280,A 0.000,B 0.000,C 90.000,E1 86.331} C_DIS
LIN {X -0.042,Y -563.405,Z 929.270,A 0.000,B 0.000,C 90.000,E1 84.666} C_DIS
LIN {X -0.137,Y -563.771,Z 929.258,A 0.000,B 0.000,C 90.000,E1 82.470} C_DIS
LIN {X 0.265,Y -564.282,Z 929.247,A 0.000,B 0.000,C 90.000,E1 80.500} C_DIS
LIN {X -0.170,Y -565.185,Z 929.235,A 0.000,B 0.000,C 90.000,E1 78.342} C_DIS
LIN {X 0.124,Y -565.982,Z 929.228,A 0.000,B 0.000,C 90.000,E1 76.937} C_DIS
LIN {X 0.180,Y -567.005,Z 929.218,A 0.000,B 0.000,C 90.000,E1 75.283} C_DIS
LIN {X 0.081,Y -567.780,Z 929.211,A 0.000,B 0.000,C 90.000,E1 73.921} C_DIS
LIN {X -0.231,Y -568.635,Z 929.202,A 0.000,B 0.000,C 90.000,E1 72.308} C_DIS
LIN {X -0.167,Y -569.359,Z 929.193,A 0.000,B 0.000,C 90.000,E1 70.659} C_DIS
LIN {X -0.051,Y -569.671,Z 929.188,A 0.000,B 0.000,C 90.000,E1 69.826} C_DIS
LIN {X 0.241,Y -570.222,Z 929.179,A 0.000,B 0.000,C 90.000,E1 68.156} C_DIS
LIN {X 0.025,Y -570.496,Z 929.170,A 0.000,B 0.000,C 90.000,E1 66.538} C_DIS
LIN {X -0.022,Y -570.705,Z 929.162,A 0.000,B 0.000,C 90.000,E1 65.177} C_DIS
LIN {X 0.072,Y -570.958,Z 929.151,A 0.000,B 0.000,C 90.000,E1 63.256} C_DIS
LIN {X -0.163,Y -570.980,Z 929.142,A 0.000,B 0.000,C 90.000,E1 61.641} C_DIS
LIN {X -0.300,Y -570.990,Z 929.132,A 0.000,B 0.000,C 90.000,E1 59.744} C_DIS
LIN {X 0.195,Y -570.895,Z 929.124,A 0.000,B 0.000,C 90.000,E1 58.329} C_DIS
LIN {X -0.101,Y -570.450,Z 929.117,A 0.000,B 0.000,C 90.000,E1 56.993} C_DIS
LIN {X 0.089,Y -570.011,Z 929.111,A 0.000,B 0.000,C 90.000,E1 55.881} C_DIS
LIN {X -0.190,Y -569.385,Z 929.104,A 0.000,B 0.000,C 90.000,E1 54.815} C_DIS
LIN {X -0.012,Y -568.669,Z 929.098,A 0.000,B 0.000,C 90.000,E1 53.703} C_DIS
LIN {X 0.035,Y -567.640,Z 929.092,A 0.000,B 0.000,C 90.000,E1 52.603} C_DIS
LIN {X 0.051,Y -566.767,Z 929.088,A 0.000,B 0.000,C 90.000,E1 51.778} C_DIS
LIN {X -0.044,Y -565.758,Z 929.083,A 0.000,B 0.000,C 90.000,E1 50.964} C_DIS
LIN {X 0.321,Y -564.156,Z 929.077,A 0.000,B 0.000,C 90.000,E1 49.828} C_DIS
LIN {X 0.100,Y -563.294,Z 929.074,A 0.000,B 0.000,C 90.000,E1 49.299} C_DIS
LIN {X -0.031,Y -561.758,Z 929.069,A 0.000,B 0.000,C 90.000,E1 48.485} C_DIS
LIN {X 0.189,Y -560.024,Z 929.065,A 0.000,B 0.000,C 90.000,E1 47.634} C_DIS
LIN {X -0.064,Y -558.797,Z 929.062,A 0.000,B 0.000,C 90.000,E1 47.106} C_DIS
LIN {X 0.165,Y -555.827,Z 929.056,A 0.000,B 0.000,C 90.000,E1 45.972} C_DIS
LIN {X 0.266,Y -554.200,Z 929.052,A 0.000,B 0.000,C 90.000,E1 45.405} C_DIS
LIN {X 0.007,Y -551.451,Z 929.048,A 0.000,B 0.000,C 90.000,E1 44.595} C_DIS
LIN {X 0.077,Y -549.449,Z 929.045,A 0.000,B 0.000,C 90.000,E1 44.028} C_DIS
LIN {X 0.164,Y -546.154,Z 929.040,A 0.000,B 0.000,C 90.000,E1 43.176} C_DIS
LIN {X -0.005,Y -544.370,Z 929.038,A 0.000,B 0.000,C 90.000,E1 42.771} C_DIS
LIN {X 0.007,Y -541.835,Z 929.035,A 0.000,B 0.000,C 90.000,E1 42.204} C_DIS
LIN {X -0.180,Y -538.353,Z 929.031,A 0.000,B 0.000,C 90.000,E1 41.515} C_DIS
LIN {X 0.184,Y -535.382,Z 929.027,A 0.000,B 0.000,C 90.000,E1 40.906} C_DIS
LIN {X 0.178,Y -532.185,Z 929.024,A 0.000,B 0.000,C 90.000,E1 40.334} C_DIS
LIN {X -0.117,Y -526.066,Z 929.019,A 0.000,B 0.000,C 90.000,E1 39.358} C_DIS
LIN {X -0.035,Y -521.494,Z 929.015,A 0.000,B 0.000,C 90.000,E1 38.624} C_DIS
LIN {X 0.191,Y -517.668,Z 929.011,A 0.000,B 0.000,C 90.000,E1 38.016} C_DIS
LIN {X 0.110,Y -510.497,Z 929.006,A 0.000,B 0.000,C 90.000,E1 36.996} C_DIS
LIN {X -0.129,Y -503.738,Z 929.001,A 0.000,B 0.000,C 90.000,E1 36.137} C_DIS
LIN {X 0.062,Y -497.851,Z 928.997,A 0.000,B 0.000,C 90.000,E1 35.391} C_DIS
LIN {X -0.171,Y -492.574,Z 928.993,A 0.000,B 0.000,C 90.000,E1 34.818} C_DIS
LIN {X 0.138,Y -487.117,Z 928.990,A 0.000,B 0.000,C 90.000,E1 34.199} C_DIS
LIN {X 0.138,Y -481.413,Z 928.987,A 0.000,B 0.000,C 90.000,E1 33.627} C_DIS
LIN {X 0.098,Y -474.474,Z 928.983,A 0.000,B 0.000,C 90.000,E1 32.959} C_DIS
LIN {X 0.080,Y -465.682,Z 928.979,A 0.000,B 0.000,C 90.000,E1 32.163} C_DIS
LIN {X -0.043,Y -456.666,Z 928.974,A 0.000,B 0.000,C 90.000,E1 31.386} C_DIS
LIN {X 0.069,Y -444.412,Z 928.969,A 0.000,B 0.000,C 90.000,E1 30.335} C_DIS
LIN {X 0.223,Y -424.373,Z 928.959,A 0.000,B 0.000,C 90.000,E1 28.615} C_DIS
LIN {X 0.079,Y -409.365,Z 928.952,A 0.000,B 0.000,C 90.000,E1 27.257} C_DIS
LIN {X 0.218,Y -400.565,Z 928.947,A 0.000,B 0.000,C 90.000,E1 26.360} C_DIS
LIN {X 0.138,Y -395.564,Z 928.943,A 0.000,B 0.000,C 90.000,E1 25.796} C_DIS
LIN {X -0.164,Y -392.186,Z 928.941,A 0.000,B 0.000,C 90.000,E1 25.335} C_DIS
LIN {X -0.026,Y -390.088,Z 928.938,A 0.000,B 0.000,C 90.000,E1 24.847} C_DIS
LIN {X 0.117,Y -389.677,Z 928.936,A 0.000,B 0.000,C 90.000,E1 24.515} C_DIS
LIN {X -0.210,Y -389.013,Z 928.934,A 0.000,B 0.000,C 90.000,E1 24.207} C_DIS
LIN {X 0.003,Y -388.785,Z 928.930,A 0.000,B 0.000,C 90.000,E1 23.462} C_DIS
LIN {X 0.175,Y -389.510,Z 928.923,A 0.000,B 0.000,C 90.000,E1 22.025} C_DIS
LIN {X 0.013,Y -393.023,Z 928.903,A 0.000,B 0.000,C 90.000,E1 18.489} C_DIS
LIN {X -0.077,Y -395.907,Z 928.889,A 0.000,B 0.000,C 90.000,E1 16.024} C_DIS
LIN {X 0.039,Y -398.175,Z 928.879,A 0.000,B 0.000,C 90.000,E1 14.245} C_DIS
LIN {X 0.146,Y -402.771,Z 928.862,A 0.000,B 0.000,C 90.000,E1 11.074} C_DIS
LIN {X -0.167,Y -406.648,Z 928.848,A 0.000,B 0.000,C 90.000,E1 8.681} C_DIS
LIN {X -0.135,Y -411.642,Z 928.833,A 0.000,B 0.000,C 90.000,E1 5.910} C_DIS
LIN {X -0.007,Y -417.801,Z 928.816,A 0.000,B 0.000,C 90.000,E1 2.808} C_DIS
LIN {X 0.161,Y -424.680,Z 928.799,A 0.000,B 0.000,C 90.000,E1 359.771} C_DIS
LIN {X -0.048,Y -428.009,Z 928.791,A 0.000,B 0.000,C 90.000,E1 358.453} C_DIS
LIN {X 0.092,Y -430.105,Z 928.788,A 0.000,B 0.000,C 90.000,E1 357.764} C_DIS
LIN {X 0.128,Y -430.745,Z 928.787,A 0.000,B 0.000,C 90.000,E1 357.593} C_DIS
LIN {X 0.161,Y -431.568,Z 928.786,A 0.000,B 0.000,C 90.000,E1 357.421} C_DIS
LIN {X -0.155,Y -434.576,Z 928.783,A 0.000,B 0.000,C 90.000,E1 356.963} C_DIS
LIN {X 0.149,Y -436.556,Z 928.782,A 0.000,B 0.000,C 90.000,E1 356.674} C_DIS
LIN {X -0.037,Y -441.119,Z 928.780,A 0.000,B 0.000,C 90.000,E1 356.331} C_DIS
LIN {X 0.161,Y -448.504,Z 928.778,A 0.000,B 0.000,C 90.000,E1 355.927} C_DIS
LIN {X 0.158,Y -460.701,Z 928.774,A 0.000,B 0.000,C 90.000,E1 355.355} C_DIS
LIN {X -0.179,Y -470.639,Z 928.772,A 0.000,B 0.000,C 90.000,E1 354.894} C_DIS
LIN {X -0.064,Y -483.949,Z 928.768,A 0.000,B 0.000,C 90.000,E1 354.204} C_DIS
LIN {X -0.087,Y -487.289,Z 928.767,A 0.000,B 0.000,C 90.000,E1 354.033} C_DIS
LIN {X -0.267,Y -497.231,Z 928.764,A 0.000,B 0.000,C 90.000,E1 353.514} C_DIS
LIN {X 0.028,Y -506.817,Z 928.761,A 0.000,B 0.000,C 90.000,E1 352.932} C_DIS
LIN {X -0.059,Y -516.289,Z 928.758,A 0.000,B 0.000,C 90.000,E1 352.356} C_DIS
LIN {X -0.169,Y -525.330,Z 928.754,A 0.000,B 0.000,C 90.000,E1 351.781} C_DIS
LIN {X 0.135,Y -534.306,Z 928.751,A 0.000,B 0.000,C 90.000,E1 351.084} C_DIS
LIN {X 0.142,Y -541.444,Z 928.747,A 0.000,B 0.000,C 90.000,E1 350.500} C_DIS
LIN {X -0.093,Y -548.121,Z 928.744,A 0.000,B 0.000,C 90.000,E1 349.926} C_DIS
LIN {X 0.000,Y -553.487,Z 928.741,A 0.000,B 0.000,C 90.000,E1 349.398} C_DIS
LIN {X -0.080,Y -558.542,Z 928.738,A 0.000,B 0.000,C 90.000,E1 348.870} C_DIS
LIN {X 0.160,Y -566.633,Z 928.733,A 0.000,B 0.000,C 90.000,E1 347.881} C_DIS
LIN {X -0.174,Y -571.990,Z 928.729,A 0.000,B 0.000,C 90.000,E1 347.229} C_DIS
LIN {X 0.313,Y -578.848,Z 928.724,A 0.000,B 0.000,C 90.000,E1 346.228} C_DIS
LIN {X -0.053,Y -583.304,Z 928.720,A 0.000,B 0.000,C 90.000,E1 345.589} C_DIS
LIN {X -0.083,Y -589.949,Z 928.714,A 0.000,B 0.000,C 90.000,E1 344.519} C_DIS
LIN {X -0.021,Y -595.926,Z 928.708,A 0.000,B 0.000,C 90.000,E1 343.449} C_DIS
LIN {X 0.296,Y -601.324,Z 928.702,A 0.000,B 0.000,C 90.000,E1 342.362} C_DIS
LIN {X 0.210,Y -605.253,Z 928.698,A 0.000,B 0.000,C 90.000,E1 341.583} C_DIS
LIN {X 0.090,Y -610.239,Z 928.692,A 0.000,B 0.000,C 90.000,E1 340.550} C_DIS
LIN {X 0.293,Y -613.847,Z 928.688,A 0.000,B 0.000,C 90.000,E1 339.752} C_DIS
LIN {X 0.280,Y -618.300,Z 928.682,A 0.000,B 0.000,C 90.000,E1 338.720} C_DIS
LIN {X -0.014,Y -621.517,Z 928.678,A 0.000,B 0.000,C 90.000,E1 337.975} C_DIS
LIN {X 0.300,Y -625.490,Z 928.672,A 0.000,B 0.000,C 90.000,E1 336.922} C_DIS
LIN {X 0.076,Y -628.336,Z 928.668,A 0.000,B 0.000,C 90.000,E1 336.177} C_DIS
LIN {X -0.100,Y -631.883,Z 928.662,A 0.000,B 0.000,C 90.000,E1 335.177} C_DIS
LIN {X 0.126,Y -636.800,Z 928.654,A 0.000,B 0.000,C 90.000,E1 333.640} C_DIS
LIN {X 0.226,Y -638.428,Z 928.651,A 0.000,B 0.000,C 90.000,E1 333.127} C_DIS
LIN {X 0.087,Y -643.347,Z 928.641,A 0.000,B 0.000,C 90.000,E1 331.385} C_DIS
LIN {X 0.125,Y -645.736,Z 928.636,A 0.000,B 0.000,C 90.000,E1 330.383} C_DIS
LIN {X -0.044,Y -648.816,Z 928.629,A 0.000,B 0.000,C 90.000,E1 329.154} C_DIS
LIN {X -0.059,Y -651.422,Z 928.622,A 0.000,B 0.000,C 90.000,E1 327.916} C_DIS
LIN {X -0.373,Y -653.594,Z 928.615,A 0.000,B 0.000,C 90.000,E1 326.707} C_DIS
LIN {X 0.069,Y -654.750,Z 928.611,A 0.000,B 0.000,C 90.000,E1 325.928} C_DIS
LIN {X -0.290,Y -656.757,Z 928.603,A 0.000,B 0.000,C 90.000,E1 324.482} C_DIS
LIN {X 0.152,Y -658.323,Z 928.594,A 0.000,B 0.000,C 90.000,E1 322.970} C_DIS
LIN {X 0.176,Y -658.838,Z 928.592,A 0.000,B 0.000,C 90.000,E1 322.477} C_DIS
LIN {X -0.310,Y -660.188,Z 928.582,A 0.000,B 0.000,C 90.000,E1 320.803} C_DIS
LIN {X -0.379,Y -661.753,Z 928.571,A 0.000,B 0.000,C 90.000,E1 318.852} C_DIS
LIN {X 0.039,Y -662.644,Z 928.566,A 0.000,B 0.000,C 90.000,E1 317.838} C_DIS
LIN {X -0.001,Y -664.005,Z 928.558,A 0.000,B 0.000,C 90.000,E1 316.377} C_DIS
LIN {X -0.025,Y -664.558,Z 928.554,A 0.000,B 0.000,C 90.000,E1 315.648} C_DIS
LIN {X -0.067,Y -666.832,Z 928.539,A 0.000,B 0.000,C 90.000,E1 312.975} C_DIS
LIN {X -0.033,Y -668.487,Z 928.529,A 0.000,B 0.000,C 90.000,E1 311.272} C_DIS
LIN {X -0.404,Y -669.594,Z 928.523,A 0.000,B 0.000,C 90.000,E1 310.092} C_DIS
LIN {X 0.196,Y -670.649,Z 928.516,A 0.000,B 0.000,C 90.000,E1 308.830} C_DIS
LIN {X -0.135,Y -671.590,Z 928.509,A 0.000,B 0.000,C 90.000,E1 307.649} C_DIS
LIN {X 0.087,Y -672.172,Z 928.504,A 0.000,B 0.000,C 90.000,E1 306.664} C_DIS
LIN {X 0.188,Y -672.472,Z 928.500,A 0.000,B 0.000,C 90.000,E1 305.931} C_DIS
LIN {X 0.281,Y -673.205,Z 928.489,A 0.000,B 0.000,C 90.000,E1 303.992} C_DIS
LIN {X 0.032,Y -674.149,Z 928.478,A 0.000,B 0.000,C 90.000,E1 302.084} C_DIS
LIN {X 0.149,Y -675.800,Z 928.465,A 0.000,B 0.000,C 90.000,E1 299.667} C_DIS
